		//缩回实时检测	
		IF (enablecloseAprSw AND NOT closeAprSw) AND closeRelay  THEN
			errorStep:=2;
		END_IF
		IF PVType=PVType_Other THEN
			;// 其他PV类型的关注点
		END_IF
	END_IF
END_IF
END_ACTION

ACTION VersionLog:
(*
版本: V1.0.0.0
说明:
	1. 首个版本
	2. 含普通PV类型的控制
	3. 可配置是否有到位信号, 以及到位稳定时间
(--------------------------------------------------)
新版本: V1.0.1.0
更新时间: 2019/11/20 19:00
更新说明:
	1. 优化编写方式
	2. 修改错误编码起始位，现改为从1开始
(--------------------------------------------------)
新版本: V1.0.1.1
更新时间: 2020/03/23 23:00
更新说明:
	1. 优化报错方式
	2. 增加打开、关闭、复位和停止触发函数
(--------------------------------------------------)
新版本: V1.0.1.2
更新时间: 2020/04/22 09:50
更新说明:
	1. 增加中文报警输出
(--------------------------------------------------)
新版本: V1.0.1.3
更新时间: 2020/09/16
更新说明:
	1. 开放错误ID、错误文本信息获取接口
(--------------------------------------------------)
新版本: V1.0.1.4
更新时间: 2020/10/06
更新说明:
	1. 移除控制模式变量，增加HMI启用条件
	2. 增加外部获取打开关闭完成信号接口函数
(--------------------------------------------------)
新版本: V1.0.1.5
更新时间: 2020/10/14
更新说明:
	1. 优化代码
(--------------------------------------------------)
*)
END_ACTION

END_FUNCTION_BLOCK

// ---- POUs/Communication/PLC_PDV.TcPOU
PROGRAM PLC_PDV
VAR_INPUT
	nSocketType:UINT:=0;// socket 类型; 0 表示 server; 1 表示 client;
	sTerminalName:STRING;// 通讯对方名称 自定义
	sHost:STRING(20):='127.0.0.1';// 通讯IP地址; server时表示本地host; client时表示远程host
	nPort:UDINT:=8900;// 通讯端口号;
	bEnable:BOOL:=TRUE;// 通讯启用\禁用连接
	sSendSuffix:STRING:='';//此处可统一添加发送后缀字符 $R$N
	nQueueInterval:UDINT:=50;// 发送队列时间间隔 单位ms
	logHandleArray:ARRAY [1..5] OF POINTER TO printLogModule_EX;// log 操作 handle 数组
	logHandleArrayLength:UINT:=0;// log 操作 handle 数组长度, 不超过5
	readStateFlag:BOOL;
	readPressureFlag:BOOL;
	readPostitionFlag:BOOL;
	readSetVal:BOOL;
	pvCloseCommunication		:BOOL;// PVClose
	pvOpenCommunication			:BOOL;// PVOpen
	pvPosOrPreCommunication		:BOOL;// PV Pos:=false;Pressure:True;
	pvReadPos:INT;// 位置
	pvReadPre:INT;// 压力
END_VAR
VAR_OUTPUT
	bSendCondition	:BOOL;//可发送条件
	bSocketConnected:BOOL;//连接状态
END_VAR
VAR CONSTANT
	cNumBegin		:DINT:=1;
	cNumEnd			:DINT:=100;
END_VAR
VAR
	sendDataArray	:ARRAY [cNumBegin..cNumEnd] OF STRING(255);
	length			:DINT:=0;
	endPoint		:DINT:=cNumBegin;
	popupSendData	:STRING(255);
	//popup
	popupStep		:UINT:=0;
	popupTON1		:TON;
	popupTON2		:TON;
	iPopup			:DINT:=0;
	_PopupLength	:DINT:=0;
END_VAR
VAR
	tcpipClient					:tcpipClientModule_EX;
	tcpipServer					:tcpipServerModule_EX;////定义服务器对象
	
	tcpipSendDataBuff_Server	:STRING(255);//发送数据 Buff server
	tcpipSendDataBuff_Client	:STRING(255);//发送数据 Buff client
	
	tcpipSendDataClear			:STRING(255);//发送数据 清空
	tcpipSendData				:STRING(255);//发送数据
	
	tcpipRecDataBuff_Server		:STRING(255);//已接收数据 Buff server
	tcpipRecDataBuff_Client		:STRING(255);//已接收数据 Buff client
	
	tcpipRecDataClear			:STRING(255);//已接收数据 清空
	tcpipRecData				:STRING(255);//已接收数据
	
	tcpConnectR_Trig			:R_Trig;//初始连接上升沿
	tcpConnectF_Trig			:F_Trig;//初始连接下降沿
	registerStep				:UDINT;//ALC注册控制步
	registerTON					:TON;//ALC注册延时
	
	logHandleArray_index		:UINT:=1;
END_VAR
VAR
	bTrig_Start:BOOL;
	rTrig_Start:R_TRIG;
	tTrig_Start:TON;
	
	bTrig_Stop:BOOL;
	rTrig_Stop:R_TRIG;
	tTrig_Stop:TON;
	
	bTrig_Reset:BOOL;
	rTrig_Reset:R_TRIG;
	tTrig_Reset:TON;
	
	
	bTrig_Init:BOOL;
	rTrig_Init:R_TRIG;
	
	bTrig_All_Home:BOOL;
	rTrig_All_Home:R_TRIG;
	
	bTrig_Z_Safe:BOOL;
	rTrig_Z_Safe:R_TRIG;
	
	bTrig_P_Pos_:BOOL;
	rTrig_P_Pos_:R_TRIG;
	nTrig_P_Pos_TrayNum:UINT:=1;
	nTrig_P_Pos_RowNum:UINT:=1;
	
	bTrig_Move_P_:BOOL;
	rTrig_Move_P_:R_TRIG;
	nTrig_Move_P_TrayNum:UINT:=1;
	nTrig_Move_P_RowNum:UINT:=1;
	nTrig_Move_P_PosNum:UINT:=1;
	findposstart	:INT;
	findposend		:INT;
	find_pos		:INT;
	recStrTemp		:STRING(255);
END_VAR


CASE nSocketType OF
0://TCPIP server
	tcpipServer(
		sSrvNetId:= , 
		sLocalHost:=sHost , 
		nLocalPort:=nPort , 
		bStartConnect:=bEnable , 
		tcpipSDataLen:=TO_UDINT(LEN(tcpipSendDataBuff_Server)) , 
		tcpipSData:=ADR(tcpipSendDataBuff_Server) , 
		bSend:= , 
		tcpipRecDataLen:=SIZEOF(tcpipRecDataBuff_Server) , 
		tcpipRecData:=ADR(tcpipRecDataBuff_Server) , 
		bAccepted=> , 
		bSendBusy=> , 
		bRecData=> );
	bSendCondition:=tcpipServer.bAccepted AND NOT tcpipServer.bSendBusy;
	//TCPIP连接
	bSocketConnected:=tcpipServer.bAccepted;
	IF NOT tcpipServer.bAccepted THEN
		length:=0;
		endPoint:=cNumBegin;
	END_IF
	tcpConnectR_Trig(CLK:=tcpipServer.bAccepted);
	tcpConnectF_Trig(CLK:=tcpipServer.bAccepted);

1://TCPIP client
	tcpipClient(
		sSrvNetId:= , 
		sRemoteHost:=sHost , 
		nRemotePort:=nPort , 
		bStartConnect:=bEnable , 
		tcpipSDataLen:=TO_UDINT(LEN(tcpipSendDataBuff_Client)) , 
		tcpipSData:=ADR(tcpipSendDataBuff_Client) , 
		bSend:= , 
		tcpipRecDataLen:=SIZEOF(tcpipRecDataBuff_Client) , 
		tcpipRecData:=ADR(tcpipRecDataBuff_Client) , 
		bConnected=> , 
		bSendBusy=> , 
		bRecData=> );
	bSendCondition:=tcpipClient.bConnected AND NOT tcpipClient.bSendBusy;
	//TCPIP连接
	bSocketConnected:=tcpipClient.bConnected;
	IF NOT tcpipClient.bConnected THEN
		length:=0;
		endPoint:=cNumBegin;
	END_IF
	tcpConnectR_Trig(CLK:=tcpipClient.bConnected);
	tcpConnectF_Trig(CLK:=tcpipClient.bConnected);
END_CASE

IF tcpConnectR_Trig.Q THEN
	FOR logHandleArray_index:=1 TO logHandleArrayLength DO
		logHandleArray[logHandleArray_index]^.append(CONCAT(sTerminalName, ' has been connected'));
	END_FOR
	registerStep:=10;
END_IF
IF tcpConnectF_Trig.Q THEN
	FOR logHandleArray_index:=1 TO logHandleArrayLength DO
		logHandleArray[logHandleArray_index]^.append(CONCAT(sTerminalName, ' has been disconnected'));
	END_FOR
	registerStep:=0;
END_IF
//数据接收处理
CASE nSocketType OF
0://TCPIP server
	IF tcpipServer.bRecData THEN
		tcpipRecData:=tcpipRecDataBuff_Server;//buff转存
		tcpipRecDataBuff_Server:=tcpipRecDataClear;//转存之后清空buff
		dataProcessing();
	END_IF
1://TCPIP client
	IF tcpipClient.bRecData THEN
		tcpipRecData:=tcpipRecDataBuff_Client;//buff转存
		tcpipRecDataBuff_Client:=tcpipRecDataClear;//转存之后清空buff
		dataProcessing();
	END_IF
END_CASE


popup();

CASE registerStep OF
0:
	//Ready
END_CASE

METHOD appendSend : BOOL
VAR_INPUT
	str			:STRING(255);
END_VAR
VAR
	suffix					:STRING;
	strTemp_appendSend		:STRING(255);
END_VAR

IF endPoint>(cNumEnd-1) THEN
	RETURN;
END_IF
suffix:=sSendSuffix;//此处可统一添加发送后缀字符 $R$N

strTemp_appendSend:=CONCAT(str,suffix);
sendDataArray[endPoint]:=strTemp_appendSend;

endPoint:=endPoint+1;
length:=endPoint-cNumBegin;
END_METHOD

METHOD dataProcessing : BOOL
VAR_INPUT
END_VAR
VAR
END_VAR
FOR logHandleArray_index:=1 TO logHandleArrayLength DO
	CASE nSocketType OF
	0://TCPIP server
	//	logHandleArray[logHandleArray_index]^.append(CONCAT(CONCAT(CONCAT('Recevie From ', sTerminalName), ' -- '),tcpipRecData));
	1://TCPIP client
	//	logHandleArray[logHandleArray_index]^.append(CONCAT(CONCAT(CONCAT('Recevie From ', sTerminalName), ' -- '),tcpipRecData));
	END_CASE
END_FOR
findposend:=0;
find_pos:=0;
IF MID(tcpipRecData,4,1)='i:30' THEN
	readStateFlag:=TRUE;
	CASE STRING_TO_INT(MID(tcpipRecData,1,6)) OF // 2:Pos 3:Close 4:Open 5:Pressur 6:Hold 7:Learn 8:interlock Open 9:interLock Closed
		2:
			pvPosOrPreCommunication:=FALSE;
			pvCloseCommunication:=FALSE;
			pvOpenCommunication:=FALSE;
		3:
			pvPosOrPreCommunication:=FALSE;
			pvCloseCommunication:=TRUE;
			pvOpenCommunication:=FALSE;
		4:
			pvPosOrPreCommunication:=FALSE;
			pvCloseCommunication:=FALSE;
			pvOpenCommunication:=TRUE;
		5:
			pvPosOrPreCommunication:=TRUE;
			pvCloseCommunication:=FALSE;
			pvOpenCommunication:=FALSE;
		ELSE
			pvPosOrPreCommunication:=FALSE;
			pvCloseCommunication:=FALSE;
			pvOpenCommunication:=FALSE;
	END_CASE
END_IF
IF MID(tcpipRecData,2,1)='A:' THEN
	readPostitionFlag:=TRUE;
	pvReadPos:=STRING_TO_INT(MID(tcpipRecData,6,3));
END_IF
IF MID(tcpipRecData,2,1)='P:' THEN
	readPressureFlag:=TRUE;
	pvReadPre:=STRING_TO_INT(MID(tcpipRecData,8,3));
	IF pvReadPre<0 THEN
		pvReadPre:=0;
	END_IF
END_IF
END_METHOD

METHOD PRIVATE popup : BOOL
VAR_INPUT
END_VAR
CASE popupStep OF
0:
	IF length>0 AND bSendCondition THEN
		_PopupLength:=length;
		popupSendData:=sendDataArray[cNumBegin];
		FOR iPopup:=cNumBegin TO (_PopupLength-1) DO
			sendDataArray[iPopup]:=sendDataArray[iPopup+1];
		END_FOR
		endPoint:=endPoint-1;
		length:=endPoint-cNumBegin;
		sendData(popupSendData);//此处是调用信息发送
		popupStep:=10;
	END_IF
10:
	popupTON2(IN:=NOT popupTON2.Q, PT:=T#2S);
	IF NOT bSendCondition OR popupTON2.Q THEN
		popupTON2(IN:=FALSE);
		popupStep:=11;
	END_IF
11:
	IF bSendCondition THEN
		popupStep:=12;
	END_IF
	popupTON1(IN:=FALSE);
12:
	//popupTON1(IN:=NOT popupTON1.Q,PT:=T#10MS);
	popupTON1(IN:=NOT popupTON1.Q,PT:=TO_TIME(nQueueInterval));
	IF popupTON1.Q THEN
		popupStep:=0;
	END_IF
END_CASE
END_METHOD

METHOD ReadPosition : BOOL
VAR_INPUT
END_VAR
VAR
END_VAR
appendSend('A:$N');
END_METHOD

METHOD ReadPressure : BOOL
VAR_INPUT
END_VAR
VAR
END_VAR
appendSend('P:$N');
END_METHOD

METHOD ReadSetVal : BOOL
VAR_INPUT
END_VAR
VAR
END_VAR
appendSend('i:38$N');
END_METHOD

METHOD ReadState : BOOL
VAR_INPUT
END_VAR
VAR
END_VAR
appendSend('i:30$N');
END_METHOD

METHOD PRIVATE sendData : BOOL
VAR_INPUT
	dataStruct	:STRING(255);
END_VAR
IF bSendCondition AND bEnable THEN
	tcpipSendData:=dataStruct;
	
	CASE nSocketType OF
	0://TCPIP server
		tcpipSendDataBuff_Server:=tcpipSendData;
		tcpipSendData:=tcpipSendDataClear;	
		tcpipServer.bSend:=TRUE;
	1://TCPIP client
		tcpipSendDataBuff_Client:=tcpipSendData;
		tcpipSendData:=tcpipSendDataClear;	
		tcpipClient.bSend:=TRUE;
	END_CASE
	
	FOR logHandleArray_index:=1 TO logHandleArrayLength DO
		CASE nSocketType OF
		0://TCPIP server
			//logHandleArray[logHandleArray_index]^.append(CONCAT(CONCAT(CONCAT('Send To ', sTerminalName), ' -- '),tcpipSendDataBuff_Server));
		1://TCPIP client
			//logHandleArray[logHandleArray_index]^.append(CONCAT(CONCAT(CONCAT('Send To ', sTerminalName), ' -- '),tcpipSendDataBuff_Client));
		END_CASE
	END_FOR
END_IF
END_METHOD

METHOD WriteAccessMode : BOOL
VAR_INPUT
	mode:INT;// 0:Local  1:Remote  2:锁定远程操作，无法通过服务端口更改为本地
END_VAR
CASE mode OF
	0:
		appendSend('c:0100$N');
	1:
		appendSend('c:0101$N');
	2:
		appendSend('c:0102$N');
	ELSE
		appendSend('c:0102$N');
END_CASE
END_METHOD

METHOD WriteCloseValve : BOOL
VAR_INPUT

END_VAR
VAR

END_VAR

appendSend('C:$N');
END_METHOD

METHOD WriteHold : BOOL
VAR_INPUT
END_VAR
appendSend('O:$N');
END_METHOD

METHOD WriteLearn : BOOL
VAR_INPUT
	positon:REAL;
	point:INT;
END_VAR
VAR
	intTemp:DINT;
	intTemp1:DINT;
	intTemp2:DINT;
	intTemp3:DINT;
	intTemp4:DINT;
	intTemp5:DINT;
	intTemp6:DINT;
	intTemp7:DINT;
	intTemp8:DINT;
	str:STRING;
END_VAR
str:='L:';
intTemp:=LREAL_TO_DINT(positon*EXPT(10,point));
intTemp8:=LREAL_TO_INT(FLOOR(intTemp/10000000));
str:=CONCAT(str,DINT_TO_STRING(intTemp8));
intTemp7:=LREAL_TO_INT(FLOOR(intTemp/1000000 MOD 10));
str:=CONCAT(str,DINT_TO_STRING(intTemp7));
intTemp6:=LREAL_TO_INT(FLOOR(intTemp/100000 MOD 10));
str:=CONCAT(str,DINT_TO_STRING(intTemp6));
intTemp5:=LREAL_TO_INT(FLOOR(intTemp/10000 MOD 10));
str:=CONCAT(str,DINT_TO_STRING(intTemp5));
intTemp4:=LREAL_TO_INT(FLOOR(intTemp/1000 MOD 10));
str:=CONCAT(str,DINT_TO_STRING(intTemp4));
intTemp3:=LREAL_TO_INT(FLOOR(intTemp/100 MOD 10));
str:=CONCAT(str,DINT_TO_STRING(intTemp3));
intTemp2:=LREAL_TO_INT(FLOOR(intTemp/10 MOD 10));
str:=CONCAT(str,DINT_TO_STRING(intTemp2));
intTemp1:=LREAL_TO_INT(FLOOR(intTemp MOD 10));
str:=CONCAT(str,DINT_TO_STRING(intTemp1));
str:=CONCAT(str,'$N');
appendSend(str);
END_METHOD

METHOD WriteOpenValve : BOOL
VAR_INPUT
END_VAR
appendSend('O:$N');
END_METHOD

METHOD WritePositionControl : BOOL
VAR_INPUT
	pressure:REAL;
	point:INT;
END_VAR
VAR
	intTemp:DINT;
	intTemp1:DINT;
	intTemp2:DINT;
	intTemp3:DINT;
	intTemp4:DINT;
	intTemp5:DINT;
	intTemp6:DINT;
	str:STRING;
END_VAR
str:='R:';
intTemp:=LREAL_TO_DINT(pressure*EXPT(10,point));
intTemp6:=LREAL_TO_INT(FLOOR(intTemp/100000 MOD 10));
str:=CONCAT(str,DINT_TO_STRING(intTemp6));
intTemp5:=LREAL_TO_INT(FLOOR(intTemp/10000 MOD 10));
str:=CONCAT(str,DINT_TO_STRING(intTemp5));
intTemp4:=LREAL_TO_INT(FLOOR(intTemp/1000 MOD 10));
str:=CONCAT(str,DINT_TO_STRING(intTemp4));
intTemp3:=LREAL_TO_INT(FLOOR(intTemp/100 MOD 10));
str:=CONCAT(str,DINT_TO_STRING(intTemp3));
intTemp2:=LREAL_TO_INT(FLOOR(intTemp/10 MOD 10));
str:=CONCAT(str,DINT_TO_STRING(intTemp2));
intTemp1:=LREAL_TO_INT(FLOOR(intTemp MOD 10));
str:=CONCAT(str,DINT_TO_STRING(intTemp1));
str:=CONCAT(str,'$N');
appendSend(str);
END_METHOD

METHOD WritePressureAlignment : BOOL
VAR_INPUT
	pressure:REAL;
	point:INT;
END_VAR
VAR
	intTemp:DINT;
	intTemp1:DINT;
	intTemp2:DINT;
	intTemp3:DINT;
	intTemp4:DINT;
	intTemp5:DINT;
	intTemp6:DINT;
	intTemp7:DINT;
	intTemp8:DINT;
	str:STRING;
END_VAR
str:='c:6002';
intTemp:=LREAL_TO_DINT(pressure*EXPT(10,point));
intTemp8:=LREAL_TO_INT(FLOOR(intTemp/10000000));
str:=CONCAT(str,DINT_TO_STRING(intTemp8));
intTemp7:=LREAL_TO_INT(FLOOR(intTemp/1000000 MOD 10));
str:=CONCAT(str,DINT_TO_STRING(intTemp7));
intTemp6:=LREAL_TO_INT(FLOOR(intTemp/100000 MOD 10));
str:=CONCAT(str,DINT_TO_STRING(intTemp6));
intTemp5:=LREAL_TO_INT(FLOOR(intTemp/10000 MOD 10));
str:=CONCAT(str,DINT_TO_STRING(intTemp5));
intTemp4:=LREAL_TO_INT(FLOOR(intTemp/1000 MOD 10));
str:=CONCAT(str,DINT_TO_STRING(intTemp4));
intTemp3:=LREAL_TO_INT(FLOOR(intTemp/100 MOD 10));
str:=CONCAT(str,DINT_TO_STRING(intTemp3));
intTemp2:=LREAL_TO_INT(FLOOR(intTemp/10 MOD 10));
str:=CONCAT(str,DINT_TO_STRING(intTemp2));
intTemp1:=LREAL_TO_INT(FLOOR(intTemp MOD 10));
str:=CONCAT(str,DINT_TO_STRING(intTemp1));
str:=CONCAT(str,'$N');
appendSend(str);
END_METHOD

METHOD WritePressureControl : BOOL
VAR_INPUT
	pressure:REAL;
	point:INT;
END_VAR
VAR
	intTemp:DINT;
	intTemp1:DINT;
	intTemp2:DINT;
	intTemp3:DINT;
	intTemp4:DINT;
	intTemp5:DINT;
	intTemp6:DINT;
	intTemp7:DINT;
	intTemp8:DINT;
	str:STRING;
END_VAR
str:='S:';
intTemp:=LREAL_TO_DINT(pressure*EXPT(10,point));
intTemp8:=LREAL_TO_INT(FLOOR(intTemp/10000000));
str:=CONCAT(str,DINT_TO_STRING(intTemp8));
intTemp7:=LREAL_TO_INT(FLOOR(intTemp/1000000 MOD 10));
str:=CONCAT(str,DINT_TO_STRING(intTemp7));
intTemp6:=LREAL_TO_INT(FLOOR(intTemp/100000 MOD 10));
str:=CONCAT(str,DINT_TO_STRING(intTemp6));
intTemp5:=LREAL_TO_INT(FLOOR(intTemp/10000 MOD 10));
str:=CONCAT(str,DINT_TO_STRING(intTemp5));
intTemp4:=LREAL_TO_INT(FLOOR(intTemp/1000 MOD 10));
str:=CONCAT(str,DINT_TO_STRING(intTemp4));
intTemp3:=LREAL_TO_INT(FLOOR(intTemp/100 MOD 10));
str:=CONCAT(str,DINT_TO_STRING(intTemp3));
intTemp2:=LREAL_TO_INT(FLOOR(intTemp/10 MOD 10));
str:=CONCAT(str,DINT_TO_STRING(intTemp2));
intTemp1:=LREAL_TO_INT(FLOOR(intTemp MOD 10));
str:=CONCAT(str,DINT_TO_STRING(intTemp1));
str:=CONCAT(str,'$N');
appendSend(str);
END_METHOD

METHOD WriteZero : BOOL
VAR_INPUT
		

END_VAR
appendSend('Z:$N');
END_METHOD

END_PROGRAM

// ---- POUs/BaseModule/TcpIpModule_EX/serverModule_EX/tcpipServerModule_EX.TcPOU
//可实现TCPIP Server 数据的收发
FUNCTION_BLOCK tcpipServerModule_EX
VAR_INPUT
	sSrvNetId			:T_AmsNetId:='';
	sLocalHost			:STRING(20):='';//服务器的IP地址
	nLocalPort			:UDINT:=5000;//服务器的端口号
	bStartConnect		:BOOL:=TRUE;//可实现外部控制服务器的重新连接
//Send
	tcpipSDataLen		:UDINT;//待发送数据长度--外部传递进来
	tcpipSData			:POINTER TO BYTE;//待发送数据源----外部以指针的形式传递进来
	bSend				:BOOL:=FALSE;//数据发送触发信号
//Receive
	tcpipRecDataLen		:UDINT;//已接收数据长度--外部传递进来
	tcpipRecData		:POINTER TO BYTE;//已接收数据源--外部以指针的形式传递进来(ADR函数)
END_VAR

VAR_OUTPUT
//Connect
	bAccepted			:BOOL:=FALSE;//表示客户端连接状态
//Send
	bSendBusy			:BOOL:=FALSE;//数据发送中
//Receive
	bRecData			:BOOL:=FALSE;//数据接收有效信号,上升沿有效
END_VAR

VAR
//Listen
	createStep			:UINT:=0;
	socketListenFB		:FB_SocketListen;(*TCP/IP Sever建立Listen功能块*)
	hListener			:T_HSOCKET;(*TCP/IP的监听句柄*)
	createDelayTime		:TIME:=T#500MS;
	createDelayTon		:TON;
	createCheckTime		:TIME:=T#1000MS;
	createCheckTon		:TON;
//Accept
	socketAcceptFB		:FB_SocketAccept;	(*TCP/IP Accept功能块*)
	hSocket				:T_HSOCKET;(*TCP/IP的句柄*)
//Send
	socketSendFB		:FB_SocketSend;	(*TCP/IP的Send功能块*)
	sendDataTempLen		:UDINT;//待发送数据缓存 长度
	sendDataTemp		:POINTER TO BYTE;//待发送数据缓存
	sendStep			:UINT:=0;
//Receive
	recStep				:UINT:=0;
	socketReceiveFB		:FB_SocketReceive;(*TCP/IP的Receive功能块*)
	recDelayTime		:TIME:=T#1S;
	recDelayTon			:TON;
//Close
	socketCloseFB		:FB_SocketClose;(*TCP/IP的Close连接的功能块*)	
END_VAR

create();
receive();
send();
socketCloseFB(
	sSrvNetId:=sSrvNetId,
	hSocket:=,
	bExecute:=FALSE);

METHOD ascii2String : STRING(g_nMaxByte_Server)
VAR_INPUT
	byteArr:ARRAY [1..g_nMaxByte_Server] OF BYTE;
END_VAR
VAR
	i:UINT;
	strTemp:STRING(g_nMaxByte_Server);
END_VAR
FOR i:=1 TO g_nMaxByte_Server DO
	strTemp:=concat(strTemp,F_ToCHR(c:=byteArr[i]));
END_FOR
ascii2string:=strTemp;
END_METHOD

METHOD PRIVATE close : BOOL
VAR_INPUT
END_VAR
//关闭hSocket这个端口的连接
socketCloseFB(
	sSrvNetId:=sSrvNetId,
	hSocket:=hSocket, 
	bExecute:=TRUE, 			//TCP/IP端口关闭的执行位
	tTimeout:=T#1S,
	bBusy=>,
	bError=>,
	nErrId=>);
socketCloseFB(
	sSrvNetId:=sSrvNetId,
	hSocket:=,
	bExecute:=FALSE);
hSocket.handle:=0;
bAccepted:=FALSE;
END_METHOD

METHOD PRIVATE closeListen : BOOL
VAR_INPUT
END_VAR
//关闭 监听 hListener 这个端口
socketCloseFB(
	sSrvNetId:=sSrvNetId,
	hSocket:=hListener, 
	bExecute:=TRUE, 			//TCP/IP端口关闭的执行位
	tTimeout:=,
	bBusy=>,
	bError=>,
	nErrId=>);
socketCloseFB(
	sSrvNetId:=sSrvNetId,
	hSocket:=,
	bExecute:=FALSE);
END_METHOD

METHOD PRIVATE create : BOOL
VAR_INPUT
END_VAR

VAR
END_VAR

CASE createStep OF
0:
	IF socketListenFB.bExecute OR bAccepted THEN
		RETURN;
	END_IF
	socketListenFB(
	   sSrvNetId:=sSrvNetId,
	   sLocalHost:=sLocalHost,
	   nLocalPort:=nLocalPort,
	   bExecute:=FALSE);
	socketCloseFB(
		sSrvNetId:=sSrvNetId,
		hSocket:=hListener, 
		bExecute:=TRUE, 			//TCP/IP端口关闭的执行位
		tTimeout:=T#1S,
		bBusy=>,
		bError=>,
		nErrId=>);
	createStep:=createStep+1;
1:
	createStep:=createStep+1;
2:
	createStep:=createStep+1;
3:
	socketListenFB(
		sSrvNetId:=sSrvNetId,
		sLocalHost:=sLocalHost,
		nLocalPort:=nLocalPort,
		bExecute:=TRUE,
		tTimeout:=T#1S,
		bBusy=>,
		bError=>,
		nErrId=>,
		hListener=>hListener);
	IF NOT socketListenFB.bBusy THEN
		IF socketListenFB.bError (*AND socketListenFB.nErrId<>32771*)THEN
			createStep:=createStep+1;
		ELSE
			//Listen
			createStep:=50;
			socketAcceptFB(
				sSrvNetId:=sSrvNetId,
				hListener:=hListener,		//TCP/IP的监听句柄
				bExecute:=FALSE);	
		END_IF
	END_IF
	createDelayTon(IN:=FALSE);

4://delay
	createDelayTon(IN:=NOT createDelayTon.Q ,PT:=createDelayTime);
	IF createDelayTon.Q THEN
		createDelayTon(IN:=FALSE);
		createStep:=createStep+1;
		socketListenFB(
			sSrvNetId:=sSrvNetId,
			sLocalHost:=sLocalHost,
			nLocalPort:=nLocalPort,
			bExecute:=FALSE);
	END_IF
5:
	createStep:=0;
	close();
	
50:	
	createStep:=51;
	close();
51:
	socketAcceptFB(
		sSrvNetId:=sSrvNetId, 
		hListener:=hListener,//TCP/IP的监听句柄
		bExecute:=TRUE,//TCP/IP接受连接请求的执行位
		tTimeout:=T#1S, 
		bAccepted=>bAccepted,
		bBusy=> , 
		bError=> , 
		nErrId=> , 
		hSocket=>hSocket );//获取的TCP/IP句柄 AND socketAcceptFB.bBusy
	IF (bAccepted AND hSocket.handle<>0) (*OR NOT bStartConnect*) THEN
		socketListenFB(
			sSrvNetId:=sSrvNetId,
			sLocalHost:=sLocalHost,
			nLocalPort:=nLocalPort,
			bExecute:=FALSE);
		createStep:=100;
	END_IF
	IF NOT bStartConnect THEN
		close();
		createStep:=100;
	END_IF
	socketAcceptFB(
		sSrvNetId:=sSrvNetId,
		hListener:=hListener,
		bExecute:=FALSE);
	createCheckTon(IN:=FALSE);

100:
	createCheckTon(IN:=NOT bAccepted OR NOT bStartConnect, PT:=createCheckTime);
	IF createCheckTon.Q THEN
		createStep:=50;
		createCheckTon(IN:=FALSE);
	END_IF
END_CASE
END_METHOD

METHOD PRIVATE receive : BOOL
VAR_INPUT
END_VAR
VAR
	recDataClear		:POINTER TO BYTE;//已接收数据源--外部以指针的形式传递进来(ADR函数)
END_VAR

CASE recStep OF
0:
	IF hSocket.handle>0 AND bAccepted THEN
		recStep:=10;
	END_IF

10:
	bRecData:=FALSE;
	socketReceiveFB(
			sSrvNetId:=sSrvNetId,
			hSocket:=hSocket,
			cbLen:= tcpipRecDataLen,
			pDest:= tcpipRecData,
			bExecute:= TRUE,
			tTimeout:=T#1S,
			bBusy=>,
			bError=>,
			nErrId=>,
			nRecBytes=>);
	
	IF (NOT socketReceiveFB.bBusy) THEN
		recStep:=20;
	END_IF
20:
	socketReceiveFB(sSrvNetId:=sSrvNetId,hSocket:=hSocket,bExecute :=FALSE);
	IF (NOT socketReceiveFB.bBusy) THEN
		IF (socketReceiveFB.bError) THEN
			close();//关闭socket
			recStep:=110;
		ELSE
			IF socketReceiveFB.nRecBytes>0 THEN
				tcpipRecData:=recDataClear;//清空缓存数据
				bRecData:=TRUE;
			END_IF
			recStep:=10;//继续接收通道数据
		END_IF
	END_IF

110:
	recDelayTon(IN:=NOT recDelayTon.Q ,PT:=recDelayTime);
	IF recDelayTon.Q THEN
		recDelayTon(IN:=FALSE);
		recStep:=recStep+10;
	END_IF
120:
	recStep:=0;	
END_CASE
END_METHOD

METHOD PRIVATE send : BOOL
VAR_INPUT
END_VAR

VAR
END_VAR

CASE sendStep OF
0:
	IF bAccepted THEN
		bSendBusy:=FALSE;
		socketSendFB(hSocket:=hSocket,bExecute :=FALSE);
		IF bSend THEN
			sendStep:=10;
			sendDataTempLen:=tcpipSDataLen;
			sendDataTemp:=tcpipSData;
			bSendBusy:=TRUE;
			bSend:=FALSE;
		END_IF
	END_IF
10:
	socketSendFB(
			sSrvNetId:=sSrvNetId, 
			hSocket:=hSocket , 
			cbLen:= sendDataTempLen,
			pSrc:= sendDataTemp, 
			bExecute:= TRUE,
			tTimeout:= T#1S, 
			bBusy=> , 
			bError=> , 
			nErrId=> );
	
	IF NOT socketSendFB.bBusy THEN
		sendStep:=sendStep+10;
	END_IF
20:
	sendStep:=sendStep+10;
30:
	bSendBusy:=FALSE;
	bSend:=FALSE;
	sendStep:=0;
END_CASE
END_METHOD

METHOD string2ASCII : ARRAY [1..g_nMaxByte_Server] OF BYTE
VAR_INPUT
	str:STRING(g_nMaxByte_Server);
END_VAR
VAR
	i:DINT;
	byteTemp:ARRAY [1..g_nMaxByte_Server] OF BYTE;
	strB:STRING(1);
	strTemp:STRING(g_nMaxByte_Server);
END_VAR

strTemp:=str;
FOR i:=1 TO g_nMaxByte_Server DO
	strB:=LEFT(strTemp,1);
	strTemp:=DELETE(strTemp,1,1);
	byteTemp[i]:=F_ToASC(str:=strB);
END_FOR
string2ASCII:=byteTemp;
END_METHOD

ACTION VersionLog:
(*
版本: V1.0.0.0
说明:
	1. 首个版本
(**************************************************)
版本: V1.0.0.1
说明:
	1. 更新close函数，关闭连接后清零连接句柄
(**************************************************)
版本: V1.0.0.2
说明:
	1. 更新cread函数，处理无法接受新连接的bug
(**************************************************)
*)
END_ACTION

END_FUNCTION_BLOCK

// ---- POUs/BaseModule/ActionModule/RFModule/RFModule.TcPOU
(*
--报错编号0: 无报错
--报错编号1: openend Error
--报错编号2: close Error
*)
FUNCTION_BLOCK RFModule
VAR_IN_OUT
	WarmHMI					:WARMStruct;
	NoteHMI					:NoteStruct;
	operatorLog				:printLogModule_EX;
END_VAR
VAR_INPUT
	HMIItf						:RFHMIStruts;// 每个RF对象都关联了一个HMI
	RFTYPE						:RFType:=RFType_Default;// 设置RF的类型
	real_TimeMonitor			:BOOL:=TRUE;//实时状态检测
	co_control					:BOOL;// 共同计时
	open						:BOOL:=FALSE;//启动触发信号
	openCondition				:BOOL:=TRUE;//启动条件
	close						:BOOL:=FALSE;//停止触发信号
	closeCondition				:BOOL:=TRUE;//停止条件
	reset						:BOOL:=FALSE;//复位信号
	readCondition				:BOOL:=TRUE;//读取条件
	stop						:BOOL:=FALSE;//停止信号
	power						:BOOL:=TRUE;// RF动作后是否关闭继电器得电状态, TRUE--保持得电,FALSE--断开得电
	enable						:BOOL:=TRUE;// RF禁用条件
	//ctrlMode					:ControlMode:=ControlMode.eManualCtrMode;//eManualCtrMode or eAutoCtrMode
	hmiEN						:BOOL:=TRUE;//HMI 启用条件
	serialExcute				:BOOL;// RS485、232开始一次参数读取
	
	errorDelayTime				:TIME:=T#100S;//分子泵感应器感应超时
	
	ACCMaxtime					:TIME:=T#20S;// RF加速最大时间 启动过程
	DCCMaxtime					:TIME:=T#20S;// RF减速最大时间 停止过程
	
	doneDelayTimeShortopenend	:TIME:=T#100MS;//  RF启动感应到位延时_伸出
	doneDelayTimeShortcloseract	:TIME:=T#50MS;//  RF感应到位延时_收回
	doneDelayTimeLongopenend	:TIME:=T#500MS;//  RF感应到位延时_伸出
	doneDelayTimeLongcloseract	:TIME:=T#50MS;// RF感应到位延时_收回
	errorID						:UDINT:=0;// RF错误报警分配的起始ID
	nameTXT						:STRING(255):='';// RF名字
	
	AlmAprSw					:BOOL:=FALSE;// RF报警感应器信号,需要链接到实际的IO点
	ErrorAprSw					:BOOL:=FALSE;// RF报错感应器信号,需要链接到实际的IO点
	enableOpenAprSw				:BOOL:=TRUE;// 启用启动感应器,针对只有一个传感器的 RF
	enableCloseAprSw			:BOOL:=TRUE;// 启用停止感应器,针对只有一个传感器的 RF
	runTime						: LINT;// 运行时间
	mainPower					:BOOL;// RF主电源
	temperature					:REAL;// RF温度
	current						:REAL;// RF电流
	vol							:REAL;// RF电压
	serialSlaveID				:UINT;// RF ID
	serialError					:BOOL;// RF通讯错误
	setpower					:UDINT;// 设定功率	
	settime						:UDINT;// 设定时间
	noteWTXT_open				:WSTRING(255):="";// RF打开动作NoteTXT 中文
	noteWTXT_close				:WSTRING(255):="";// RF关闭动作NoteTXT 中文
	controlMode					:INT:=0;// 0 手动，1 Analog，2 RS232
	outputMode					:INT:=0;// 0 continuous，1 pulse
	outputState					:INT:=0;// 0 Stop,1 Start
	alarmState					:INT:=0;// 0 No Error,1 Error
	setpowerRead				:UDINT:=0;// 读取设置的功率值
	forwardpower				:UDINT;// 实际功率	
	reflectedpower				:UDINT;// 反馈功率
	maxpower					:UDINT;// 设置的最大功率值
END_VAR
VAR_OUTPUT
	note_open				:BOOL;// 开条件不满足提示
	note_close				:BOOL;// 关条件不满足提示
	openRelay				:BOOL:=FALSE;// RF启动执行继电器,需要链接到实际的IO点
	closeRelay				:BOOL:=FALSE;// RF停止执行继电器,需要链接到实际的IO点
	resetRelay				:BOOL:=FALSE;// RF复位执行继电器,需要链接到实际的IO点	
	rematime				:UDINT;// 剩余时间
	busy					:BOOL;// RFusy状态
	openbusy				:BOOL;// RF开动作Busy状态
	closebusy				:BOOL;// RF关动作Busy状态
	readbusy				:BOOL;// RF循环读取Busy状态
	done					:BOOL;// RF动作Done状态
	readdone					:BOOL;// RF动作Done状态
	opendone				:BOOL;// RF动作伸出完成
	closedone				:BOOL;// RF动作收回完成
	setpointdone			:BOOL;
	readerror			    :BOOL;// RF动作error状态
	error					:BOOL;// RF动作error状态
	errID					:UDINT;// RF动作errID
	errTXT					:STRING(255):='';// RF动作errTXT
	errWTXT					:WSTRING(255):="";// RF动作errTXT 中文
END_VAR
	
VAR	
	readAndWriteLock:BOOL;
	runTON					: TON;
	openErrorDelayTon		:Ton;
	openDoneDelayTon		:Ton;
	closeErrorDelayTon		:Ton;
	closeDoneDelayTon		:Ton;
	
	extendTrigRAlc			:R_Trig;//上升沿触发
	runTimeClearR			:R_Trig;//上升沿触发
	
	openendTrigRAlc			:R_Trig;//上升沿触发
	
	singleControltempR			:R_Trig;//上升沿触发
	singleControlR			:R_Trig;//上升沿触发
	singleControlF			:F_Trig;//上升沿触发
	
	openendTrigR1			:R_Trig;//上升沿触发
	openendTrigR1_Aiko		:R_Trig;//上升沿触发
	closeractTrigR1			:R_Trig;//上升沿触发
	resetTrigR1				:R_Trig;//上升沿触发
	stopTrigR1				:R_Trig;//上升沿触发
	powerTrigR1				:R_Trig;//上升沿触发
	
	openStep				:UINT:=0;
	closeStep				:UINT:=0;
	errorStep				:UINT:=0;
	readStep				:UINT:=0;
	
	resetRelayTON			:TON;
	resetRelayTONTime		:TIME:=T#2S;
	
	writeStep				:UINT:=0;
	writeMaxStep			:UINT:=0;
	
	notBusyMonitorDelayTon:TON;//动作不切换时，延迟检测
	notBusyMonitorDelayTime:TIME:=T#2S;//动作不切换延迟检测时间
	firstPower			    :BOOL:=TRUE;//首次上电标志位
	firstPowerTON			:TON;
	AccFTrig:F_TRIG;//检测加速信号下降延
	NormalRTrig:R_TRIG;//匀速上升沿
	DccFTrig:F_TRIG;// 检测减速信号下降延
	noteTON_P:tON;            // 操作提示标志位延时继电器
	noteTON_N:tON;            // 操作提示标志位延时继电器
	noteRTrig_P:R_TRIG;          // 操作提示
	noteRTrig_N:R_TRIG;          // 操作提示
	powerTon:TON;
	readTon1:TON;
	readTon2:TON;
	readTon3:TON;
	t1:TON;
	t2:TON;
	writeTON:TON;
	writeMaxTON:TON;
	readTON:TON;
	readErrorTimes:UINT:=0;
END_VAR

Init_ACT();
Error_ACT();
Open_ACT();
Close_ACT();
Reset_ACT();
Error_ACT();
Read_ACT();
WritePower_ACT();
WriteMaxPower_ACT();

(*
触发缩回动作，成功触发返回TRUE，触发失败返回FALSE
*)
METHOD Act_Close : BOOL
VAR_INPUT
END_VAR
IF enable AND closeCondition THEN// AND NOT busy
	Act_Close:=close:=TRUE;
ELSE
	Act_Close:=FALSE;
END_IF
END_METHOD

(*
触发伸出动作，成功触发返回TRUE，触发失败返回FALSE
*)
METHOD Act_Open : BOOL
VAR_INPUT
END_VAR
IF enable AND openCondition THEN// AND NOT busy
	Act_Open:=open:=TRUE;
ELSE
	Act_Open:=FALSE;
END_IF
END_METHOD

(*
触发复位报警动作，成功触发返回TRUE，触发失败返回FALSE
*)
METHOD Act_Reset : BOOL
VAR_INPUT
END_VAR
Act_Reset:=reset:=TRUE;
END_METHOD

(*
触发发送动作，成功触发返回TRUE，触发失败返回FALSE
*)
METHOD Act_SerialSend : BOOL
VAR_INPUT
END_VAR
IF TRUE THEN
	Act_SerialSend:=serialExcute:=TRUE;
ELSE
	Act_SerialSend:=FALSE;
END_IF
END_METHOD

METHOD Act_SetPoint : BOOL
VAR_INPUT
	setpoint:UDINT;
	_settime:UDINT;
	con_ctr:BOOL;
END_VAR
VAR_OUTPUT
	outTime:UDINT;
END_VAR
setpower:=HMIItf.setpower:=setpoint;
settime:=HMIItf.settime:=outTime:=_settime;
co_control:=con_ctr;
Act_Open();
END_METHOD

(*
触发停止输出动作，成功触发返回TRUE，触发失败返回FALSE
*)
METHOD Act_Stop : BOOL
VAR_INPUT
END_VAR
Act_Stop:=stop:=TRUE;
END_METHOD

(*
触发缩回动作，成功触发返回TRUE，触发失败返回FALSE
*)
METHOD Act_Write : BOOL
VAR_INPUT
END_VAR
IF writeStep<10 AND NOT readAndWriteLock THEN
	writeStep:=10;
	readAndWriteLock:=TRUE;
END_IF
END_METHOD

(*
触发缩回动作，成功触发返回TRUE，触发失败返回FALSE
*)
METHOD Act_Write_1 : BOOL
VAR_INPUT
END_VAR
IF writeStep<10 AND readAndWriteLock THEN
	writeStep:=10;
	readAndWriteLock:=TRUE;
END_IF
END_METHOD

ACTION Close_ACT:
//分子泵--close 触发
IF close AND NOT closeCondition THEN
	note_open:=FALSE;
	note_close:=TRUE;
	NoteHMI.showFlag:=TRUE;
	NoteHMI.showText:='';
	NoteHMI.showText:=CONCAT(NoteHMI.showText,nameTXT);
	NoteHMI.showText:=CONCAT(NoteHMI.showText,' Close Condition Not Satisfied!');
	operatorLog.append(CONCAT(nameTXT,' Close Not Done '));
END_IF
IF close AND enable AND closeCondition AND closeStep<20 THEN// AND NOT busy
	note_open:=FALSE;
	note_close:=FALSE;
	busy:=TRUE;
	writeStep:=0;
	writeMaxStep:=0;
	closebusy:=TRUE;
	openbusy:=FALSE;
	open:=FALSE;
	// searial_send(0)**************************************
	opendone:=FALSE;
	closedone:=FALSE;
	openStep:=0;
	closeStep:=10;
	readAndWriteLock:=TRUE;
	PLC_PowerRF.WriteStop();
	operatorLog.append(CONCAT(nameTXT,' Close Done '));
	//errorStep:=0;
END_IF
close:=FALSE;

CASE closeStep OF
0:
	//ready
	
10:
	IF readStep<10 AND writeStep<10 AND writeMaxStep<10 THEN
		closeErrorDelayTon(IN:=FALSE);
		closeDoneDelayTon(IN:=FALSE);
		closeRelay:=TRUE;
		PLC_PowerRF.WriteStop();
		openRelay:=FALSE;
		closeStep:=15;
		t2(IN:=FALSE);
	END_IF
15:
	t2(IN:=TRUE,PT:=T#0.2S);
	IF t2.Q THEN
		t2(IN:=FALSE);
		readAndWriteLock:=FALSE;
		PLC_PowerRF.WriteStop();
		closeStep:=20;
		busy:=FALSE;
	END_IF
20:// DCC与ACC一样，只不过ACC在Open逻辑；DCC 在Close逻辑里；  DCC=forwardpower<setpoint
	closeErrorDelayTon(IN:=(NOT (forwardpower=0 AND reflectedpower=0 AND rematime=0)),PT:=errorDelayTime);
	IF closeErrorDelayTon.Q THEN
		//done:=FALSE;
		opendone:=FALSE;
		closedone:=FALSE;
		errorStep:=2;
		closeStep:=40;
		RETURN;
	END_IF
	IF enablecloseAprSw THEN
		closeDoneDelayTon(IN:=(forwardpower=0 AND reflectedpower=0 AND rematime=0),PT:=doneDelayTimeShortcloseract);
	END_IF
	IF closeDoneDelayTon.Q THEN
		closeErrorDelayTon(IN:=FALSE);
		closeDoneDelayTon(IN:=FALSE);
		closeStep:=30;
	END_IF
30:
	busy:=FALSE;
	closebusy:=FALSE;
	openbusy:=FALSE;
	//done:=TRUE;
	opendone:=FALSE;
	closedone:=TRUE;
	errorStep:=0;
	closeStep:=0;
	readAndWriteLock:=FALSE;
	t2(IN:=FALSE);
40:
	busy:=FALSE;
	closebusy:=FALSE;
	openbusy:=FALSE;
	closeStep:=0;
	readAndWriteLock:=FALSE;
	t2(IN:=FALSE);
END_CASE
END_ACTION

ACTION Error_ACT:
CASE errorStep OF
	0:
		error:=FALSE;
		errID:=0;
		errTXT:='';
 (*
	1:
		error:=TRUE;
		errID:=errorID+errorStep;
		errTXT:=CONCAT(STR1:=nameTXT,STR2:=' Extend Error!');
		errWTXT:=WCONCAT(STR1:=TO_WSTRING(nameTXT),STR2:=" 伸出(打开)错误");
	2:
		error:=TRUE;
		errID:=errorID+errorStep;
		errTXT:=CONCAT(STR1:=nameTXT,STR2:=' Retract Error!');
		errWTXT:=WCONCAT(STR1:=TO_WSTRING(nameTXT),STR2:=" 缩回(关闭)错误");
		*)
	1..6:
		error:=TRUE;
		errID:=getErrID(errorStep);
		errTXT:=getErrTXT(errorStep);
		errWTXT:=getErrWTXT(errorStep);
END_CASE
END_ACTION

METHOD Get_Done_Close : BOOL
VAR_INPUT
END_VAR
Get_Done_Close:=closedone;
END_METHOD

METHOD Get_Done_Open : BOOL
VAR_INPUT
END_VAR
Get_Done_Open:=opendone;
END_METHOD

METHOD getErrID : UDINT
VAR_INPUT
	errID					:UDINT;//取值范围1~2
END_VAR
VAR
	nErrID					:UDINT;
END_VAR
nErrID:=errorID+errID;

getErrID:=nErrID;
END_METHOD

METHOD getErrTXT : STRING(255)
VAR_INPUT
	errID					:UDINT;//取值范围1~2
END_VAR
VAR
	sErrTXT					:STRING(255);
END_VAR

CASE errID OF
	1:
		sErrTXT:=CONCAT(STR1:=nameTXT,STR2:=' Open(TimeOut) Error!');
	2:
		sErrTXT:=CONCAT(STR1:=nameTXT,STR2:=' Close Error!');
	3:
		sErrTXT:=CONCAT(STR1:=nameTXT,STR2:=' NormalRun Error!');
	4:
		sErrTXT:=CONCAT(STR1:=nameTXT,STR2:=' CheckCondition Error!');
	5:
		sErrTXT:=CONCAT(STR1:=nameTXT,STR2:=' ParSet Fault!');
	6:
		sErrTXT:=CONCAT(STR1:=nameTXT,STR2:=' Communication Error!');
ELSE
	sErrTXT:=CONCAT(STR1:=nameTXT,STR2:='');
END_CASE
getErrTXT:=sErrTXT;
END_METHOD

METHOD getErrWTXT : WSTRING(255)
VAR_INPUT
	errID					:UDINT;//取值范围1~16
END_VAR
VAR
	sErrTXT					:WSTRING(255);
END_VAR

CASE errID OF
	1:
		sErrTXT:=WCONCAT(STR1:=TO_WSTRING(nameTXT),STR2:=" RF启动错误");
	2:
		sErrTXT:=WCONCAT(STR1:=TO_WSTRING(nameTXT),STR2:=" RF停止错误");
	3:
		sErrTXT:=WCONCAT(STR1:=TO_WSTRING(nameTXT),STR2:=" RF正常运行出现异常情况");
	4:
		sErrTXT:=WCONCAT(STR1:=TO_WSTRING(nameTXT),STR2:=" 检测到条件异常，关机处理");
	5:
		sErrTXT:=WCONCAT(STR1:=TO_WSTRING(nameTXT),STR2:=" 参数设置有误");
	6:
		sErrTXT:=WCONCAT(STR1:=TO_WSTRING(nameTXT),STR2:=" 通讯异常");
		
ELSE
	sErrTXT:=WCONCAT(STR1:=TO_WSTRING(nameTXT),STR2:="");
END_CASE
getErrWTXT:=sErrTXT;
END_METHOD

ACTION Init_ACT:
done:=(opendone OR closedone);
powerTon(IN:=mainPower,PT:=T#10S);
IF AlmAprSw AND powerTon.Q THEN
	errorStep:=5;
END_IF
IF readerror OR NOT readCondition AND firstPowerTON.Q THEN
	errorStep:=6;
END_IF
error:=error OR serialError OR NOT mainPower OR AlmAprSw;
InitHMI_ACT();
manualCtrl_ACT();
IF (error OR AlmAprSw OR ErrorAprSw OR NOT openCondition) AND openRelay THEN
	stop:=TRUE;
	busy:=FALSE;
	openRelay:=FALSE;
END_IF

noteTON_P(IN:=note_open,PT:=T#0.1S);
noteRTrig_P(CLK:=noteTON_P.Q);
IF noteRTrig_P.Q THEN
//	gLog_Note.append_EX(noteWTXT_Open);
END_IF
noteTON_N(IN:=note_close,PT:=T#0.1S);
noteRTrig_N(CLK:=noteTON_N.Q);
IF noteRTrig_N.Q THEN
//	gLog_Note.append_EX(noteWTXT_close);
END_IF
END_ACTION

ACTION InitHMI_ACT:
HMIItf.AlmAprSw:=AlmAprSw;
HMIItf.ErrorAprSw:=ErrorAprSw;

HMIItf.temperature:=temperature;
HMIItf.current:=current;
HMIItf.vol:=vol;

HMIItf.enableOpen:=enableOpenAprSw;
HMIItf.enableClose:=enableCloseAprSw;
HMIItf.HMIEnable:=hmiEN;
HMIItf.enable:=enable;
HMIItf.done:=done;
HMIItf.busy:=busy;
HMIItf.error:=error;
HMIItf.errID:=UDINT_TO_DINT(errID);
HMIItf.errTXT:=errTXT;
HMIItf.openRelay:=openRelay;
HMIItf.resetRelay:=resetRelay;

HMIItf.power:=power;
HMIItf.nameTXT:=nameTXT;

HMIItf.runTime:=runTime;
HMIItf.opencondition:=openCondition;
HMIItf.closecondition:=closeCondition;
END_ACTION

ACTION ManualCtrl_ACT:
//HMI手动控制
//IF ctrlMode=eManualCtrMode THEN
IF hmiEN THEN
	extendTrigRAlc(CLK:=HMIItf.extendAndretract);
	IF extendTrigRAlc.Q THEN// AND NOT busy
		IF openRelay THEN// 如果启动继电器或全速，则认为已经已启动完毕
			close:=TRUE;
		END_IF
		IF NOT openRelay THEN
			open:=TRUE;
		END_IF
	END_IF
	openendTrigR1_Aiko(CLK:=HMIItf.bopen);
	IF openendTrigR1_Aiko.Q AND NOT busy AND NOT openRelay THEN
		open:=TRUE;
		close:=FALSE;
	END_IF
	IF openendTrigR1_Aiko.Q AND busy AND openRelay THEN
		close:=TRUE;
		open:=FALSE;
	END_IF
	
	singleControltempR(CLK:=HMIItf.singleControltemp);
	openendTrigR1(CLK:=HMIItf.open);
	IF openendTrigR1.Q OR (singleControltempR.Q AND NOT openRelay ) THEN// AND NOT busy
		WarmHMI.showText:='';
		WarmHMI.showFlag:=TRUE;
		WarmHMI.showText:=CONCAT(WarmHMI.showText,'Are you sure you want to Open the ');
		WarmHMI.showText:=CONCAT(WarmHMI.showText,nameTXT);
		WarmHMI.showText:=CONCAT(WarmHMI.showText,' ?');
	END_IF
	IF WarmHMI.bOK AND NOT WarmHMI.showFlag AND FIND(WarmHMI.showText,nameTXT)>0 AND FIND(WarmHMI.showText,'Open')>0 THEN
		open:=TRUE;
		WarmHMI.bOK:=FALSE;
		WarmHMI.showText:='';
		operatorLog.append(CONCAT(CONCAT(nameTXT,' Open:'),UDINT_TO_STRING(setpower)));
		operatorLog.append(CONCAT(CONCAT(nameTXT,' Open:'),UDINT_TO_STRING(settime)));
	END_IF
	IF WarmHMI.bNO AND NOT WarmHMI.showFlag AND FIND(WarmHMI.showText,nameTXT)>0 AND FIND(WarmHMI.showText,'Open')>0 THEN
		WarmHMI.bNO:=FALSE;
		WarmHMI.showText:='';
	END_IF
	
	closeractTrigR1(CLK:=HMIItf.close);
	IF closeractTrigR1.Q OR (singleControltempR.Q AND openRelay) THEN// AND NOT busy
		WarmHMI.showText:='';
		WarmHMI.showFlag:=TRUE;
		WarmHMI.showText:=CONCAT(WarmHMI.showText,'Are you sure you want to Close the ');
		WarmHMI.showText:=CONCAT(WarmHMI.showText,nameTXT);
		WarmHMI.showText:=CONCAT(WarmHMI.showText,' ?');
	END_IF
	IF WarmHMI.bOK AND NOT WarmHMI.showFlag AND FIND(WarmHMI.showText,nameTXT)>0 AND FIND(WarmHMI.showText,'Close')>0 THEN
		close:=TRUE;
		operatorLog.append(CONCAT(nameTXT,' Close'));
		WarmHMI.bOK:=FALSE;
		WarmHMI.showText:='';
	END_IF
	IF WarmHMI.bNO AND NOT WarmHMI.showFlag AND FIND(WarmHMI.showText,nameTXT)>0 AND FIND(WarmHMI.showText,'Close')>0 THEN
		WarmHMI.bNO:=FALSE;
		WarmHMI.showText:='';
	END_IF
	
	resetTrigR1(CLK:=HMIItf.reset);
	IF resetTrigR1.Q THEN// AND NOT busy
		reset:=TRUE;
	END_IF
	
	stopTrigR1(CLK:=HMIItf.stop);
	IF stopTrigR1.Q THEN// AND NOT busy
		stop:=TRUE;
	END_IF
	
	powerTrigR1(CLK:=HMIItf.power);
	IF powerTrigR1.Q THEN// AND NOT busy
		IF power THEN
			power:=FALSE;
		ELSE
			power:=TRUE;
		END_IF
	END_IF
	
END_IF
END_ACTION

ACTION Open_ACT:
//分子泵伸出--open 触发
IF open AND NOT openCondition THEN
	note_open:=TRUE;
	note_close:=FALSE;
	NoteHMI.showFlag:=TRUE;
	NoteHMI.showText:='';
	NoteHMI.showText:=CONCAT(NoteHMI.showText,nameTXT);
	NoteHMI.showText:=CONCAT(NoteHMI.showText,' Open Condition Not Satisfied!');
	operatorLog.append(CONCAT(nameTXT,' Open Not Done '));
END_IF
IF open AND enable AND openCondition AND NOT AlmAprSw AND NOT ErrorAprSw AND NOT openbusy AND mainPower AND NOT resetRelay THEN// AND NOT busy
	note_open:=FALSE;
	note_close:=FALSE;
	busy:=TRUE;
	closebusy:=FALSE;
	openbusy:=TRUE;
	close:=FALSE;
	open:=FALSE;
	done:=FALSE;
	opendone:=FALSE;
	closedone:=FALSE;
	openStep:=10;
	writeStep:=0;
	writeMaxStep:=0;
	readAndWriteLock:=TRUE;
	// searial_send(setPoint)**************************************
	closeStep:=0;
	operatorLog.append(CONCAT(nameTXT,' Open Done '));
END_IF
open:=FALSE;
runTimeClearR(CLK:=HMIItf.runTimeClear);
runTON(IN:=NOT error AND openRelay AND NOT runTON.Q, PT:=T#60S);// 1小时计数一次,启动，无报错，且全速
IF runTON.Q AND runTime<999999999999999 AND NOT runTimeClearR.Q THEN
	runTime:=runTime+1;
END_IF
IF runTimeClearR.Q THEN
	runTime:=0;
END_IF
//IF NOT openRelay AND NOT AccAprSw AND NOT DccAprSw AND NOT NormalAprSw THEN// 计数清零
//	runTime:=0;
//END_IF

CASE openStep OF
0:
	//ready
	runTON(IN:=FALSE);
	openErrorDelayTon(IN:=FALSE);
	openErrorDelayTon(IN:=FALSE);
	openDoneDelayTon(IN:=FALSE);
	t1(IN:=FALSE);
	rematime:=0;
10:
	IF setpower<1 OR (NOT co_control AND settime<1) THEN 
		open:=FALSE;
		close:=FALSE;
		openbusy:=FALSE;
		closebusy:=FALSE;
		errorStep:=5;
		openStep:=60;
	ELSE
		t1(IN:=readStep<10 AND writeStep<10 AND writeMaxStep<10,PT:=T#0.5S);
		IF t1.Q THEN
			openErrorDelayTon(IN:=FALSE);
			openDoneDelayTon(IN:=FALSE);
			openStep:=15;
			openRelay:=TRUE;
			setpointdone:=FALSE;
			Act_Write_1();
			openbusy:=TRUE;
			closebusy:=FALSE;
			closeRelay:=FALSE;
			t1(IN:=FALSE);
		END_IF
	END_IF
15:
	t1(IN:=setpointdone,PT:=T#0.1S);
	IF t1.Q THEN
		setpointdone:=FALSE;
		t1(IN:=FALSE);
		PLC_PowerRF.receiveFlag:=FALSE;
		PLC_PowerRF.WriteStart();
		openStep:=17;
	END_IF
17:
	t1(IN:=PLC_PowerRF.receiveFlag,PT:=T#0.05S);
	IF t1.Q THEN
		t1(IN:=FALSE);
		PLC_PowerRF.receiveFlag:=FALSE;
		readAndWriteLock:=FALSE;
		busy:=false;
		openStep:=20;
	END_IF
20:
	// AccAprSw可以看成是forward Power > 5 ,< set point - 5// 或者反射功率>0
	openErrorDelayTon(IN:=(NOT (ABS(forwardpower)>=0 AND reflectedpower<10 AND ABS(setpower-forwardpower)<2)),PT:=errorDelayTime);
	IF openErrorDelayTon.Q THEN
		//done:=FALSE;
		open:=FALSE;
		close:=FALSE;
		openbusy:=FALSE;
		closebusy:=FALSE;
		errorStep:=1;
		openStep:=60;
		RETURN;
	END_IF
	IF enableopenAprSw THEN
		openDoneDelayTon(IN:=ABS(forwardpower)>=0 AND reflectedpower<10 AND ABS(setpower-forwardpower)<2,PT:=doneDelayTimeShortopenend);
	END_IF
	IF openDoneDelayTon.Q THEN
		openErrorDelayTon(IN:=FALSE);
		openDoneDelayTon(IN:=FALSE);
		openStep:=30;
	END_IF
	
	//状态实时检测
	IF NOT openCondition AND (NOT closedone OR openRelay) THEN// 检测到开条件消失，强制关闭
		openRelay:=FALSE;
		errorStep:=4;
		openbusy:=FALSE;
		closebusy:=FALSE;
		openStep:=60;
	END_IF
	IF (ErrorAprSw OR AlmAprSw) AND openRelay THEN//只要报错；启动线圈启动，强锁启动信号
		openRelay:=FALSE;
		openStep:=60;/////
		errorStep:=3;
		openbusy:=FALSE;
		closebusy:=FALSE;
	END_IF
30:
	openErrorDelayTon(IN:=NOT co_control,PT:=UDINT_TO_TIME(settime*1000));// 反射调整超时时间
	rematime:=TIME_TO_UDINT(openErrorDelayTon.ET/1000);
	rematime:=settime-rematime;
	IF openErrorDelayTon.Q OR co_control THEN
		openStep:=40;
		rematime:=0;
		openErrorDelayTon(IN:=FALSE);
	END_IF
	// 状态实时检测
	IF NOT openCondition AND (NOT closedone OR openRelay) THEN//蝶阀单控，检测到开条件消失，强制关闭
		openRelay:=FALSE;
		errorStep:=4;
		openStep:=60;
		closebusy:=FALSE;
		openbusy:=FALSE;
	END_IF
	IF (ErrorAprSw OR AlmAprSw) AND openRelay THEN//只要报错；启动线圈启动，强锁启动信号
		openRelay:=FALSE;
		stop:=TRUE;
		openStep:=60;/////
		errorStep:=3;
		closebusy:=FALSE;
		openbusy:=FALSE;
	END_IF
40:
	busy:=FALSE;
	IF NOT co_control THEN
		openRelay:=FALSE;
		close:=TRUE;
	END_IF
	openStep:=50;
	openbusy:=FALSE;
	readAndWriteLock:=FALSE;
	opendone:=TRUE;
50:
	rematime:=0;
60:
	openRelay:=FALSE;
	openStep:=70;
	busy:=FALSE;
	readAndWriteLock:=FALSE;
	;//报错
	co_control:=FALSE;
	opendone:=FALSE;
END_CASE
END_ACTION

ACTION Read_ACT:
//气缸收回--read 触发
firstPowerTON(IN:=firstPower,PT:=T#10S);
readTON(IN:=NOT readAndWriteLock AND NOT busy AND  NOT readbusy AND readStep=0 AND readCondition,PT:=T#0.05S);
IF readTON.Q THEN// AND NOT busy
	readdone:=FALSE;
	readStep:=10;
	readbusy:=TRUE;
	readerror:=FALSE;
END_IF
CASE readStep OF
0:
	//ready
	readTon1(IN:=FALSE);
	readTon2(IN:=FALSE);
	readTon3(IN:=FALSE);
10:// State
	IF gICP.PowerRF.controlMode=2 THEN
		PLC_PowerRF.readStateFlag:=FALSE;
		PLC_PowerRF.ReadState();
		readStep:=readStep+10;
	ELSE
		PLC_PowerRF.readStateFlag:=FALSE;
		PLC_PowerRF.WriteRS232Mode();
		readStep:=readStep+15;
		PLC_PowerRF.receiveFlag:=FALSE;
	END_IF
20:
	IF PLC_PowerRF.readStateFlag THEN
		PLC_PowerRF.readStateFlag:=FALSE;
		// 数据处理
		readTon1(IN:=FALSE);
		readStep:=readStep+10;
		RETURN;
	END_IF
	readTon1(IN:=TRUE,PT:=T#500MS);// 超时
	IF readTon1.Q THEN
		readStep:=6000;
		readTon1(IN:=FALSE);
		readTon2(IN:=FALSE);
		RETURN;
	END_IF
25:
	IF PLC_PowerRF.receiveFlag THEN
		PLC_PowerRF.receiveFlag:=FALSE;
		// 数据处理
		readTon1(IN:=FALSE);
		readStep:=readStep+5;
		RETURN;
	END_IF
	readTon1(IN:=TRUE,PT:=T#500MS);// 超时
	IF readTon1.Q THEN
		readStep:=6000;
		readTon1(IN:=FALSE);
		readTon2(IN:=FALSE);
		RETURN;
	END_IF
30:
	readTon3(IN:=TRUE,PT:=T#0.1S);
	IF readTon3.Q THEN
		readStep:=readStep+10;
		readTon3(IN:=FALSE);
	END_IF
40:// State
	PLC_PowerRF.readStateFlag:=FALSE;
	PLC_PowerRF.ReadState();
	readStep:=readStep+10;
50:
	IF PLC_PowerRF.readStateFlag THEN
		PLC_PowerRF.readStateFlag:=FALSE;
		// 数据处理
		readTon1(IN:=FALSE);
		readStep:=readStep+10;
		RETURN;
	END_IF
	readTon1(IN:=TRUE,PT:=T#500MS);// 超时
	IF readTon1.Q THEN
		readStep:=6000;
		readTon1(IN:=FALSE);
		readTon2(IN:=FALSE);
		RETURN;
	END_IF
60:
	readStep:=90;
90:
	readTon3(IN:=TRUE,PT:=T#0.1S);
	IF readTon3.Q THEN
		readStep:=5000;
		readTon3(IN:=FALSE);
	END_IF
5000:
	readbusy:=FALSE;
	readdone:=TRUE;
	readStep:=0;
	readerror:=FALSE;
	PLC_PowerRF.ClearCom:=TRUE;
6000:
	readbusy:=FALSE;
	readdone:=TRUE;
	readStep:=0;
	readErrorTimes:=readErrorTimes+1;
	IF readErrorTimes>3 THEN
		readErrorTimes:=0;
		readerror:=TRUE;
		gICP.PowerRF.setpowerRead:=0;
		gICP.PowerRF.forwardpower:=0;
		gICP.PowerRF.reflectedpower:=0;
		gICP.PowerRF.maxpower:=0;
	END_IF
	gICP.PowerRF.controlMode:=0;
END_CASE
END_ACTION

ACTION Reset_ACT:
IF reset THEN
	IF NOT power THEN
		openRelay:=FALSE;
		closeRelay:=FALSE;
	END_IF
	note_open:=FALSE;
	note_close:=FALSE;
	IF errorStep<>0 OR  AlmAprSw OR ErrorAprSw THEN
		errorStep:=0;
		busy:=FALSE;
		closebusy:=FALSE;
		openbusy:=FALSE;
		resetRelay:=TRUE;
		readAndWriteLock:=TRUE;
		PLC_PowerRF.WriteReset();
	END_IF
	reset:=FALSE;
	note_open:=FALSE;
	note_close:=FALSE;
END_IF
resetRelayTON(IN:=resetRelay , PT:=resetRelayTONTime);
IF resetRelayTON.Q THEN
	errorStep:=0;
	busy:=FALSE;
	resetRelay:=FALSE;
	readAndWriteLock:=FALSE;
END_IF

IF stop THEN
	note_open:=FALSE;
	note_close:=FALSE;
	stop:=FALSE;
	openRelay:=FALSE;
	closeRelay:=FALSE;
	//无自锁检测说法，直接停
	openStep:=0;
	closeStep:=0;
	writeStep:=0;
	writeMaxStep:=0;
END_IF
END_ACTION

ACTION VersionLog:
(*
版本: V1.0.0.0
说明:
	1. 首个版本
	2. 含普通分子泵\泵组类型的控制
	3. 可配置是否有到位信号, 以及到位稳定时间
(--------------------------------------------------)
新版本: V1.0.1.0
更新时间: 2019/11/20 19:00
更新说明:
	1. 优化编写方式
	2. 修改错误编码起始位，现改为从1开始
(--------------------------------------------------)
新版本: V1.0.1.1
更新时间: 2020/03/23 23:00
更新说明:
	1. 优化报错方式
	2. 增加伸出、缩回、复位和停止触发函数
(--------------------------------------------------)
新版本: V1.0.1.2
更新时间: 2020/04/22 09:50
更新说明:
	1. 增加中文报警输出
(--------------------------------------------------)
新版本: V1.0.1.3
更新时间: 2020/09/16
更新说明:
	1. 开放错误ID、错误文本信息获取接口
(--------------------------------------------------)
新版本: V1.0.1.4
更新时间: 2020/10/06
更新说明:
	1. 移除控制模式变量，增加HMI启用条件
	2. 增加外部获取伸出缩回完成信号接口函数
(--------------------------------------------------)
新版本: V1.0.1.5
更新时间: 2020/10/14
更新说明:
	1. 优化代码
(--------------------------------------------------)
新版本: V2.0.1.0
更新时间: 2023/11/17
更新说明:
	1. 分子泵控制独立
(--------------------------------------------------)


*)
END_ACTION

ACTION WriteMaxPower_ACT:
//分子泵--writeMax 触发

CASE writeMaxStep OF
0:
	//ready
	writeMaxTON(IN:=FALSE);
10:
	writeMaxTON(IN:=readStep<10,PT:=T#0.1S);
	IF writeMaxTON.Q THEN
		PLC_PowerRF.ClearCom:=TRUE;
		writeMaxTON(IN:=FALSE);
		writeMaxStep:=writeMaxStep+10;
	END_IF
20:
	IF readStep<10 AND openStep<10 AND closeStep<10 AND writeMaxStep<10 THEN
		PLC_PowerRF.WriteMaxPower(gICP.PowerRF.setpower);
		PLC_PowerRF.receiveFlag:=FALSE;
		writeMaxStep:=writeMaxStep+10;
	END_IF
30:
	writeMaxTON(IN:=NOT PLC_PowerRF.receiveFlag ,PT:=T#0.5S);
	IF writeMaxTON.Q THEN
		PLC_PowerRF.receiveFlag:=FALSE;
		writeMaxTON(IN:=FALSE);
		writeMaxStep:=writeMaxStep+10;
		RETURN;
	END_IF
	IF PLC_PowerRF.receiveFlag THEN
		PLC_PowerRF.receiveFlag:=FALSE;
		writeMaxTON(IN:=FALSE);
		writeMaxStep:=writeMaxStep+10;
		RETURN;
	END_IF
40:
	writeMaxStep:=100;
100:
	writeMaxStep:=0;	
	readAndWriteLock:=FALSE;
END_CASE
END_ACTION

ACTION WritePower_ACT:
//分子泵--write 触发

CASE writeStep OF
0:
	//ready
	writeTON(IN:=FALSE);
10:
	writeTON(IN:=readStep<10,PT:=T#0.1S);
	setpointdone:=FALSE;
	IF writeTON.Q THEN
		PLC_PowerRF.ClearCom:=TRUE;
		writeTON(IN:=FALSE);
		writeStep:=writeStep+10;
	END_IF
20:
	IF readStep<10  AND writeMaxStep<10 THEN
		PLC_PowerRF.WritePower(gICP.PowerRF.setpower);
		PLC_PowerRF.receiveFlag:=FALSE;
		writeStep:=writeStep+10;
	END_IF
30:
	writeTON(IN:=NOT PLC_PowerRF.receiveFlag ,PT:=T#0.5S);
	IF writeTON.Q THEN
		PLC_PowerRF.receiveFlag:=FALSE;
		writeTON(IN:=FALSE);
		writeStep:=writeStep+10;
		setpointdone:=FALSE;
		RETURN;
	END_IF
	IF PLC_PowerRF.receiveFlag THEN
		PLC_PowerRF.receiveFlag:=FALSE;
		writeTON(IN:=FALSE);
		writeStep:=writeStep+10;
		setpointdone:=TRUE;
		RETURN;
	END_IF
40:
	writeStep:=100;
100:
	writeStep:=0;	
	readAndWriteLock:=FALSE;
END_CASE
END_ACTION

END_FUNCTION_BLOCK

// ---- POUs/Communication/PLC_PowerRF.TcPOU
PROGRAM PLC_PowerRF
VAR_INPUT
	nSocketType:UINT:=0;// socket 类型; 0 表示 server; 1 表示 client;
	sTerminalName:STRING;// 通讯对方名称 自定义
	sHost:STRING(20):='127.0.0.1';// 通讯IP地址; server时表示本地host; client时表示远程host
	nPort:UDINT:=8900;// 通讯端口号;
	bEnable:BOOL:=TRUE;// 通讯启用\禁用连接
	sSendSuffix:STRING:='';//此处可统一添加发送后缀字符 $R$N
	nQueueInterval:UDINT:=50;// 发送队列时间间隔 单位ms
	logHandleArray:ARRAY [1..5] OF POINTER TO printLogModule_EX;// log 操作 handle 数组
	logHandleArrayLength:UINT:=0;// log 操作 handle 数组长度, 不超过5
	readStateFlag:BOOL;
	ClearCom:BOOL;
	receiveFlag:BOOL;
END_VAR
VAR_OUTPUT
	bSendCondition	:BOOL;//可发送条件
	bSocketConnected:BOOL;//连接状态
END_VAR
VAR CONSTANT
	cNumBegin		:DINT:=1;
	cNumEnd			:DINT:=100;
END_VAR
VAR
	sendDataArray	:ARRAY [cNumBegin..cNumEnd] OF STRING(255);
	length			:DINT:=0;
	endPoint		:DINT:=cNumBegin;
	popupSendData	:STRING(255);
	//popup
	popupStep		:UINT:=0;
	popupTON1		:TON;
	popupTON2		:TON;
	iPopup			:DINT:=0;
	_PopupLength	:DINT:=0;
END_VAR
VAR
	tcpipClient					:tcpipClientModule_EX;
	tcpipServer					:tcpipServerModule_EX;////定义服务器对象
	
	tcpipSendDataBuff_Server	:STRING(255);//发送数据 Buff server
	tcpipSendDataBuff_Client	:STRING(255);//发送数据 Buff client
	
	tcpipSendDataClear			:STRING(255);//发送数据 清空
	tcpipSendData				:STRING(255);//发送数据
	
	tcpipRecDataBuff_Server		:STRING(255);//已接收数据 Buff server
	tcpipRecDataBuff_Client		:STRING(255);//已接收数据 Buff client
	
	tcpipRecDataClear			:STRING(255);//已接收数据 清空
	tcpipRecData				:STRING(255);//已接收数据
	
	tcpConnectR_Trig			:R_Trig;//初始连接上升沿
	tcpConnectF_Trig			:F_Trig;//初始连接下降沿
	registerStep				:UDINT;//ALC注册控制步
	registerTON					:TON;//ALC注册延时
	
	logHandleArray_index		:UINT:=1;
END_VAR
VAR
	bTrig_Start:BOOL;
	rTrig_Start:R_TRIG;
	tTrig_Start:TON;
	
	bTrig_Stop:BOOL;
	rTrig_Stop:R_TRIG;
	tTrig_Stop:TON;
	
	bTrig_Reset:BOOL;
	rTrig_Reset:R_TRIG;
	tTrig_Reset:TON;
	
	
	bTrig_Init:BOOL;
	rTrig_Init:R_TRIG;
	
	bTrig_All_Home:BOOL;
	rTrig_All_Home:R_TRIG;
	
	bTrig_Z_Safe:BOOL;
	rTrig_Z_Safe:R_TRIG;
	
	bTrig_P_Pos_:BOOL;
	rTrig_P_Pos_:R_TRIG;
	nTrig_P_Pos_TrayNum:UINT:=1;
	nTrig_P_Pos_RowNum:UINT:=1;
	
	bTrig_Move_P_:BOOL;
	rTrig_Move_P_:R_TRIG;
	nTrig_Move_P_TrayNum:UINT:=1;
	nTrig_Move_P_RowNum:UINT:=1;
	nTrig_Move_P_PosNum:UINT:=1;
	findposstart	:INT;
	findposend		:INT;
	find_pos		:INT;
	recStrTemp		:STRING(255);
END_VAR


CASE nSocketType OF
0://TCPIP server
	tcpipServer(
		sSrvNetId:= , 
		sLocalHost:=sHost , 
		nLocalPort:=nPort , 
		bStartConnect:=bEnable , 
		tcpipSDataLen:=TO_UDINT(LEN(tcpipSendDataBuff_Server)) , 
		tcpipSData:=ADR(tcpipSendDataBuff_Server) , 
		bSend:= , 
		tcpipRecDataLen:=SIZEOF(tcpipRecDataBuff_Server) , 
		tcpipRecData:=ADR(tcpipRecDataBuff_Server) , 
		bAccepted=> , 
		bSendBusy=> , 
		bRecData=> );
	bSendCondition:=tcpipServer.bAccepted AND NOT tcpipServer.bSendBusy;
	//TCPIP连接
	bSocketConnected:=tcpipServer.bAccepted;
	IF NOT tcpipServer.bAccepted THEN
		length:=0;
		endPoint:=cNumBegin;
	END_IF
	tcpConnectR_Trig(CLK:=tcpipServer.bAccepted);
	tcpConnectF_Trig(CLK:=tcpipServer.bAccepted);

1://TCPIP client
	tcpipClient(
		sSrvNetId:= , 
		sRemoteHost:=sHost , 
		nRemotePort:=nPort , 
		bStartConnect:=bEnable , 
		tcpipSDataLen:=TO_UDINT(LEN(tcpipSendDataBuff_Client)) , 
		tcpipSData:=ADR(tcpipSendDataBuff_Client) , 
		bSend:= , 
		tcpipRecDataLen:=SIZEOF(tcpipRecDataBuff_Client) , 
		tcpipRecData:=ADR(tcpipRecDataBuff_Client) , 
		bConnected=> , 
		bSendBusy=> , 
		bRecData=> );
	bSendCondition:=tcpipClient.bConnected AND NOT tcpipClient.bSendBusy;
	//TCPIP连接
	bSocketConnected:=tcpipClient.bConnected;
	IF NOT tcpipClient.bConnected THEN
		length:=0;
		endPoint:=cNumBegin;
	END_IF
	tcpConnectR_Trig(CLK:=tcpipClient.bConnected);
	tcpConnectF_Trig(CLK:=tcpipClient.bConnected);
END_CASE
IF ClearCom THEN
	length:=0;
	endPoint:=cNumBegin;
	ClearCom:=FALSE;
END_IF
IF tcpConnectR_Trig.Q THEN
	FOR logHandleArray_index:=1 TO logHandleArrayLength DO
		logHandleArray[logHandleArray_index]^.append(CONCAT(sTerminalName, ' has been connected'));
	END_FOR
	registerStep:=10;
END_IF
IF tcpConnectF_Trig.Q THEN
	FOR logHandleArray_index:=1 TO logHandleArrayLength DO
		logHandleArray[logHandleArray_index]^.append(CONCAT(sTerminalName, ' has been disconnected'));
	END_FOR
	registerStep:=0;
END_IF
//数据接收处理
CASE nSocketType OF
0://TCPIP server
	IF tcpipServer.bRecData THEN
		tcpipRecData:=tcpipRecDataBuff_Server;//buff转存
		tcpipRecDataBuff_Server:=tcpipRecDataClear;//转存之后清空buff
		dataProcessing();
	END_IF
1://TCPIP client
	IF tcpipClient.bRecData THEN
		tcpipRecData:=tcpipRecDataBuff_Client;//buff转存
		tcpipRecDataBuff_Client:=tcpipRecDataClear;//转存之后清空buff
		dataProcessing();
	END_IF
END_CASE


popup();

CASE registerStep OF
0:
	//Ready
END_CASE

METHOD appendSend : BOOL
VAR_INPUT
	str			:STRING(255);
END_VAR
VAR
	suffix					:STRING;
	strTemp_appendSend		:STRING(255);
END_VAR

IF endPoint>(cNumEnd-1) THEN
	RETURN;
END_IF
suffix:=sSendSuffix;//此处可统一添加发送后缀字符 $R$N

strTemp_appendSend:=CONCAT(str,suffix);
sendDataArray[endPoint]:=strTemp_appendSend;

endPoint:=endPoint+1;
length:=endPoint-cNumBegin;
END_METHOD

METHOD dataProcessing : BOOL
VAR_INPUT
END_VAR
VAR
	strTemp:STRING;
END_VAR
FOR logHandleArray_index:=1 TO logHandleArrayLength DO
	CASE nSocketType OF
	0://TCPIP server
//		logHandleArray[logHandleArray_index]^.append(CONCAT(CONCAT(CONCAT('Recevie From ', sTerminalName), ' -- '),tcpipRecData));
	1://TCPIP client
//		logHandleArray[logHandleArray_index]^.append(CONCAT(CONCAT(CONCAT('Recevie From ', sTerminalName), ' -- '),tcpipRecData));
	END_CASE
END_FOR
receiveFlag:=TRUE;
findposend:=0;
find_pos:=0;
IF MID(tcpipRecData,1,32)='$R' AND MID(tcpipRecData,1,33)='$R'  THEN
	gICP.PowerRF.controlMode:=STRING_TO_INT(MID(tcpipRecData,1,1));
	gICP.PowerRF.outputMode:=STRING_TO_INT(MID(tcpipRecData,1,2));
	gICP.PowerRF.outputState:=STRING_TO_INT(MID(tcpipRecData,1,3));
	strTemp:='';
	strTemp:=CONCAT(strTemp,(MID(tcpipRecData,2,6)));
	gICP.PowerRF.alarmState:=STRING_TO_INT(strTemp);
	strTemp:='';
	strTemp:=CONCAT(strTemp,(MID(tcpipRecData,5,9)));
	gICP.PowerRF.setpowerRead:=STRING_TO_UDINT(strTemp);
	strTemp:='';
	strTemp:=CONCAT(strTemp,(MID(tcpipRecData,5,15)));
	gICP.PowerRF.forwardpower:=STRING_TO_UDINT(strTemp);
	strTemp:='';
	strTemp:=CONCAT(strTemp,(MID(tcpipRecData,5,21)));
	gICP.PowerRF.reflectedpower:=STRING_TO_UDINT(strTemp);
	strTemp:='';
	strTemp:=CONCAT(strTemp,(MID(tcpipRecData,5,27)));
	gICP.PowerRF.maxpower:=STRING_TO_UDINT(strTemp);
	readStateFlag:=TRUE;
END_IF
END_METHOD

METHOD PRIVATE popup : BOOL
VAR_INPUT
END_VAR
CASE popupStep OF
0:
	IF length>0 AND bSendCondition THEN
		_PopupLength:=length;
		popupSendData:=sendDataArray[cNumBegin];
		FOR iPopup:=cNumBegin TO (_PopupLength-1) DO
			sendDataArray[iPopup]:=sendDataArray[iPopup+1];
		END_FOR
		endPoint:=endPoint-1;
		length:=endPoint-cNumBegin;
		sendData(popupSendData);//此处是调用信息发送
		popupStep:=10;
	END_IF
10:
	popupTON2(IN:=NOT popupTON2.Q, PT:=T#2S);
	IF NOT bSendCondition OR popupTON2.Q THEN
		popupTON2(IN:=FALSE);
		popupStep:=11;
	END_IF
11:
	IF bSendCondition THEN
		popupStep:=12;
	END_IF
	popupTON1(IN:=FALSE);
12:
	//popupTON1(IN:=NOT popupTON1.Q,PT:=T#10MS);
	popupTON1(IN:=NOT popupTON1.Q,PT:=TO_TIME(nQueueInterval));
	IF popupTON1.Q THEN
		popupStep:=0;
	END_IF
END_CASE
END_METHOD

METHOD ReadState : BOOL
VAR_INPUT
END_VAR
VAR
END_VAR
appendSend('Q$R');
END_METHOD

METHOD PRIVATE sendData : BOOL
VAR_INPUT
	dataStruct	:STRING(255);
END_VAR
IF bSendCondition AND bEnable THEN
	tcpipSendData:=dataStruct;
	
	CASE nSocketType OF
	0://TCPIP server
		tcpipSendDataBuff_Server:=tcpipSendData;
		tcpipSendData:=tcpipSendDataClear;	
		tcpipServer.bSend:=TRUE;
	1://TCPIP client
		tcpipSendDataBuff_Client:=tcpipSendData;
		tcpipSendData:=tcpipSendDataClear;	
		tcpipClient.bSend:=TRUE;
	END_CASE
	
	FOR logHandleArray_index:=1 TO logHandleArrayLength DO
		CASE nSocketType OF
		0://TCPIP server
//			logHandleArray[logHandleArray_index]^.append(CONCAT(CONCAT(CONCAT('Send To ', sTerminalName), ' -- '),tcpipSendDataBuff_Server));
		1://TCPIP client
//			logHandleArray[logHandleArray_index]^.append(CONCAT(CONCAT(CONCAT('Send To ', sTerminalName), ' -- '),tcpipSendDataBuff_Client));
		END_CASE
	END_FOR
END_IF
END_METHOD

METHOD WriteMaxPower : BOOL
VAR_INPUT
	maxpowerpoint:UDINT;
END_VAR
VAR
	str:STRING;
	_bit:UDINT;
	_ten:UDINT;
	_hundred:UDINT;
	_thousand:UDINT;
END_VAR
str:='';
_thousand:=maxpowerpoint/1000;
str:=CONCAT(str,UDINT_TO_STRING(maxpowerpoint));
//_hundred:=maxpowerpoint/100 MOD 10;
//str:=CONCAT(str,UDINT_TO_STRING(_hundred));
//_ten:=maxpowerpoint/10 MOD 10;
//str:=CONCAT(str,UDINT_TO_STRING(_ten));
//_bit:=maxpowerpoint MOD 10;
//str:=CONCAT(str,UDINT_TO_STRING(_bit));
str:=CONCAT(str,' M$R');
appendSend(str);
END_METHOD

METHOD WritePower : BOOL
VAR_INPUT
	powerpoint:UDINT;
END_VAR
VAR
	str:STRING;
	_bit:UDINT;
	_ten:UDINT;
	_hundred:UDINT;
	_thousand:UDINT;
END_VAR
str:='';
//_thousand:=powerpoint/1000;
str:=CONCAT(str,UDINT_TO_STRING(powerpoint));
//_hundred:=powerpoint/100 MOD 10;
//str:=CONCAT(str,UDINT_TO_STRING(_hundred));
//_ten:=powerpoint/10 MOD 10;
//str:=CONCAT(str,UDINT_TO_STRING(_ten));
//_bit:=powerpoint MOD 10;
//str:=CONCAT(str,UDINT_TO_STRING(_bit));
str:=CONCAT(str,' W$R');
appendSend(str);
END_METHOD

METHOD WriteReset : BOOL
VAR_INPUT
		

END_VAR
appendSend('RESET$R');
END_METHOD

METHOD WriteRS232Mode : BOOL
VAR_INPUT
		

END_VAR
appendSend('***$R');
END_METHOD

METHOD WriteStart : BOOL
VAR_INPUT
		

END_VAR
appendSend('G$R');
END_METHOD

METHOD WriteStop : BOOL
VAR_INPUT
		

END_VAR
appendSend('S$R');
END_METHOD

END_PROGRAM

// ---- POUs/BaseModule/ActionModule/chillerModule/ChillerModule_1.TcPOU
(*
--报错编号0: 无报错
--报错编号1: Extend Error
--报错编号2: Retract Error
*)
FUNCTION_BLOCK ChillerModule_1
VAR_IN_OUT
	WarmHMI					:WARMStruct;
	NoteHMI					:NoteStruct;
	operatorLog				:printLogModule_EX;
END_VAR
VAR_INPUT
	HMIItf						:ChillerModuleHMI;//每个Chiller对象都关联了一个HMI
	ChillerType				:ChillerType:=ChillerType_Default;//设置Chiller的类型, 可通过该变量修改为真空发生器
	
	real_TimeMonitor			:BOOL:=TRUE;//实时状态检测
	
	extend						:BOOL:=FALSE;//伸出触发信号
	extCondition				:BOOL:=TRUE;//伸出启停条件
	retract						:BOOL:=FALSE;//收回触发信号
	retCondition				:BOOL:=TRUE;//收回启停条件
	setPoint					:BOOL:=FALSE;//设置触发信号
	setCondition				:BOOL:=TRUE;//设置启停条件
	readPoint					:BOOL:=FALSE;// 设置读取信号
	readCondition				:BOOL:=TRUE;// 设置读取条件
	reset						:BOOL:=FALSE;//复位信号
	stop						:BOOL:=FALSE;//停止信号
	power						:BOOL:=TRUE;//Chiller动作后是否关闭继电器得电状态, TRUE--保持得电,FALSE--断开得电
	enable						:BOOL:=TRUE;//Chiller禁用条件
	//ctrlMode					:ControlMode:=ControlMode.eManualCtrMode;//eManualCtrMode or eAutoCtrMode
	hmiEN						:BOOL:=TRUE;//HMI 启用条件
	
	errorDelayTime				:TIME:=T#3000MS;//Chiller感应器感应超时
	//doneDelayTimeShort		:TIME:=T#100MS;//Chiller感应到位延时---取消使用
	//doneDelayTimeLong			:TIME:=T#500MS;//无Chiller感应到位延时---取消使用
	doneDelayTimeShortExtend	:TIME:=T#100MS;//Chiller感应到位延时_伸出
	doneDelayTimeShortRetract	:TIME:=T#100MS;//Chiller感应到位延时_收回
	doneDelayTimeLongExtend		:TIME:=T#500MS;//无Chiller感应到位延时_伸出
	doneDelayTimeLongRetract	:TIME:=T#500MS;//无Chiller感应到位延时_收回
	doneDelayTimeLongSET		:TIME:=T#500MS;//无Chiller感应到位延时_SET
	errorID						:UDINT:=0;//Chiller错误报警分配的起始ID
	nameTXT						:STRING(255):='';//Chiller名字
	
	extAprSw					:BOOL:=FALSE;//Chiller伸出感应器信号,需要链接到实际的IO点
	retAprSw					:BOOL:=FALSE;//Chiller收回感应器信号,需要链接到实际的IO点
	enableExtAprSw				:BOOL:=TRUE;//启用伸出感应器,针对只有一个传感器的Chiller
	enableRetAprSw				:BOOL:=TRUE;//启用收回感应器,针对只有一个传感器的Chiller
	
	noteWTXT_Ext				:WSTRING(255):="";//Chiller伸出动作NoteTXT 中文
	noteWTXT_Ret				:WSTRING(255):="";//Chiller缩回动作NoteTXT 中文
	pumon:BOOL;		
	uinton:BOOL;
	fault:BOOL;
	unitstoping:BOOL;
	alarmTemperatureH			:REAL:=30;
	alarmTemperatureL			:REAL:=10;
	RTD1:REAL;
	RTD2:REAL;
	setpointVal					:REAL;
END_VAR
VAR_OUTPUT
	extRelay				:BOOL:=FALSE;//Chiller伸出执行继电器,需要链接到实际的IO点
	retRelay				:BOOL:=FALSE;//Chiller收回执行继电器,需要链接到实际的IO点
	note_Ext				:BOOL:=FALSE;// 操作提示：true 伸出、打开执行无法下发
	note_Ret				:BOOL:=FALSE;// 操作提示：true 缩回、关闭执行无法下发
	note_Set				:BOOL:=FALSE;// 操作提示：true 设置参数执行无法下发
	busy					:BOOL;//Chiller动作Busy状态
	readbusy				:BOOL;
	readerror				:BOOL;
	done					:BOOL;//Chiller动作Done状态
	extdone					:BOOL;//Chiller动作伸出完成
	retdone					:BOOL;//Chiller动作收回完成
	setdone					:BOOL;//Chiller动作收回完成
	readdone				:BOOL;//Chiller动作收回完成
	error					:BOOL;//Chiller动作error状态
	errID					:UDINT;//Chiller动作errID
	errTXT					:STRING(255):='';//Chiller动作errTXT
	errWTXT					:WSTRING(255):="";//Chiller动作errTXT 中文
	sensorShow				:STRING;
END_VAR
	
VAR
	readAndWriteLock:BOOL;
	firstPower:BOOL:=TRUE;
	extErrorDelayTon		:Ton;
	extDoneDelayTon			:Ton;
	retErrorDelayTon		:Ton;
	retDoneDelayTon			:Ton;
	setErrorDelayTon		:Ton;
	setDoneDelayTon			:Ton;
	readConditionTon		:TON;
	readTon1				:TON;
	readTon2				:TON;
	
	extendTrigRAlc			:R_Trig;//上升沿触发
	
	singleControlR			:R_Trig;//上升沿触发
	singleControlF			:F_Trig;//上升沿触发
	
	setR					:R_Trig;//上升沿触发
	
	extendTrigR1			:R_Trig;//上升沿触发
	retractTrigR1			:R_Trig;//上升沿触发
	resetTrigR1				:R_Trig;//上升沿触发
	stopTrigR1				:R_Trig;//上升沿触发
	powerTrigR1				:R_Trig;//上升沿触发
	
	extStep					:UINT:=0;
	retStep					:UINT:=0;
	setStep					:UINT:=0;
	readStep				:UINT:=0;
	errorStep				:UINT:=0;
	
	notBusyMonitorDelayTon:TON;//动作不切换时，延迟检测
	notBusyMonitorDelayTime:TIME:=T#2S;//动作不切换延迟检测时间
	noteTON_P:tON;            // 操作提示标志位延时继电器
	noteTON_N:tON;            // 操作提示标志位延时继电器
	noteRTrig_P:R_TRIG;          // 操作提示
	noteRTrig_N:R_TRIG;          // 操作提示
	extRealayRtrig:R_TRIG;
	retRealayRtrig:R_TRIG;
END_VAR

// 实时读取设置的流量值以及实际反馈浏览值
// ****************************
Init_ACT();
Error_ACT();
Extend_ACT();
Retract_ACT();
Reset_ACT();
Set_ACT();
Read_ACT();
Error_ACT();
SafeMonitor_ACT();

(*
触发伸出动作，成功触发返回TRUE，触发失败返回FALSE
*)
METHOD Act_Extend : BOOL
VAR_INPUT
END_VAR
IF enable AND extCondition THEN// AND NOT busy
	Act_Extend:=extend:=TRUE;
ELSE
	Act_Extend:=FALSE;
END_IF
END_METHOD

(*
触发复位报警动作，成功触发返回TRUE，触发失败返回FALSE
*)
METHOD Act_Reset : BOOL
VAR_INPUT
END_VAR
Act_Reset:=reset:=TRUE;
END_METHOD

(*
触发缩回动作，成功触发返回TRUE，触发失败返回FALSE
*)
METHOD Act_Retract : BOOL
VAR_INPUT
END_VAR
IF enable AND retCondition THEN// AND NOT busy
	Act_Retract:=retract:=TRUE;
ELSE
	Act_Retract:=FALSE;
END_IF
END_METHOD

(*
触发停止输出动作，成功触发返回TRUE，触发失败返回FALSE
*)
METHOD Act_Stop : BOOL
VAR_INPUT
END_VAR
Act_Stop:=stop:=TRUE;
END_METHOD

ACTION Error_ACT:
CASE errorStep OF
	0:
		error:=FALSE;
		errID:=0;
		errTXT:='';
 (*
	1:
		error:=TRUE;
		errID:=errorID+errorStep;
		errTXT:=CONCAT(STR1:=nameTXT,STR2:=' Extend Error!');
		errWTXT:=WCONCAT(STR1:=TO_WSTRING(nameTXT),STR2:=" 伸出(打开)错误");
	2:
		error:=TRUE;
		errID:=errorID+errorStep;
		errTXT:=CONCAT(STR1:=nameTXT,STR2:=' Retract Error!');
		errWTXT:=WCONCAT(STR1:=TO_WSTRING(nameTXT),STR2:=" 缩回(关闭)错误");
		*)
	1..4:
		error:=TRUE;
		errID:=getErrID(errorStep);
		errTXT:=getErrTXT(errorStep);
		errWTXT:=getErrWTXT(errorStep);
END_CASE
END_ACTION

ACTION Extend_ACT:
// Chiller伸出--extend 触发
IF extend AND NOT extCondition THEN
	note_Ext:=TRUE;
	note_Ret:=FALSE;
	note_Set:=FALSE;
	NoteHMI.showFlag:=TRUE;
	NoteHMI.showText:='';
	NoteHMI.showText:=CONCAT(NoteHMI.showText,nameTXT);
	NoteHMI.showText:=CONCAT(NoteHMI.showText,' Open Condition Not Satisfied!');
	HMIItf.singleControl:=FALSE;
END_IF
IF extend AND enable AND extCondition THEN// AND NOT busy
	busy:=TRUE;
	retract:=FALSE;
	setPoint:=FALSE;
	setPoint:=FALSE;
	extdone:=FALSE;
	retdone:=FALSE;
	setdone:=FALSE;
	extStep:=10;
	retStep:=0;
	setStep:=0;
	note_Ext:=FALSE;
	note_Ret:=FALSE;
	note_Set:=FALSE;
	readAndWriteLock:=TRUE;
	//errorStep:=0;
END_IF
extend:=FALSE;
CASE extStep OF
0:
	//ready
	extErrorDelayTon(IN:=FALSE);
10:
	firstPower:=FALSE;
	extErrorDelayTon(IN:=FALSE);
	extDoneDelayTon(IN:=FALSE);
	extStep:=20;
	PLC_Chiller.readStartFlag:=FALSE;
	PLC_Chiller.WriteStart();
	extRelay:=TRUE;
	retRelay:=FALSE;
20:
	extErrorDelayTon(IN:=(NOT PLC_Chiller.readStartFlag),PT:=errorDelayTime);
	IF extErrorDelayTon.Q THEN
		//done:=FALSE;
		extdone:=FALSE;
		retdone:=FALSE;
		setdone:=FALSE;
		errorStep:=1;
		busy:=FALSE;
		readAndWriteLock:=FALSE;
		extStep:=40;
		extErrorDelayTon(IN:=FALSE);
		RETURN;
	END_IF
//	IF PLC_Chiller.readStartFlag THEN
//		extDoneDelayTon(IN:=PLC_Chiller.readStartFlag,PT:=doneDelayTimeShortExtend);
//	ELSE
//		extDoneDelayTon(IN:=NOT enableExtAprSw,PT:=doneDelayTimeLongExtend);
//	END_IF
	
	IF PLC_Chiller.readStartFlag THEN
		PLC_Chiller.readStartFlag:=FALSE;
		busy:=FALSE;
		//done:=TRUE;
		extdone:=TRUE;
		readAndWriteLock:=FALSE;
		retdone:=FALSE;
		errorStep:=0;
		IF NOT power THEN
			extRelay:=FALSE;
			retRelay:=FALSE;
		END_IF
		extStep:=30;
		extErrorDelayTon(IN:=FALSE);
	END_IF
END_CASE
END_ACTION

METHOD Get_Done_Ext : BOOL
VAR_INPUT
END_VAR
Get_Done_Ext:=extdone;
END_METHOD

METHOD Get_Done_Ret : BOOL
VAR_INPUT
END_VAR
Get_Done_Ret:=retdone;
END_METHOD

METHOD getErrID : UDINT
VAR_INPUT
	errID					:UDINT;//取值范围1~2
END_VAR
VAR
	nErrID					:UDINT;
END_VAR
nErrID:=errorID+errID;

getErrID:=nErrID;
END_METHOD

METHOD getErrTXT : STRING(255)
VAR_INPUT
	errID					:UDINT;//取值范围1~2
END_VAR
VAR
	sErrTXT					:STRING(255);
END_VAR

CASE errID OF
	1:
		sErrTXT:=CONCAT(STR1:=nameTXT,STR2:=' Extend Error!');
	2:
		sErrTXT:=CONCAT(STR1:=nameTXT,STR2:=' Retract Error!');
	3:
		sErrTXT:=CONCAT(STR1:=nameTXT,STR2:=' ParSet Error!');
	4:
		sErrTXT:=CONCAT(STR1:=nameTXT,STR2:=' State Error!');
ELSE
	sErrTXT:=CONCAT(STR1:=nameTXT,STR2:='');
END_CASE
getErrTXT:=sErrTXT;
END_METHOD

METHOD getErrWTXT : WSTRING(255)
VAR_INPUT
	errID					:UDINT;//取值范围1~16
END_VAR
VAR
	sErrTXT					:WSTRING(255);
END_VAR

CASE errID OF
	1:
		sErrTXT:=WCONCAT(STR1:=TO_WSTRING(nameTXT),STR2:=" 伸出(打开)错误");
	2:
		sErrTXT:=WCONCAT(STR1:=TO_WSTRING(nameTXT),STR2:=" 缩回(关闭)错误");
	3:
		sErrTXT:=WCONCAT(STR1:=TO_WSTRING(nameTXT),STR2:=" 参数设置错误");
ELSE
	sErrTXT:=WCONCAT(STR1:=TO_WSTRING(nameTXT),STR2:="");
END_CASE
getErrWTXT:=sErrTXT;
END_METHOD

ACTION Init_ACT:
done:=(extdone OR retdone);
InitHMI_ACT();
manualCtrl_ACT();
IF RTD1>alarmTemperatureH OR RTD1<alarmTemperatureL OR 
   RTD2>alarmTemperatureH OR RTD2<alarmTemperatureL THEN
   errorID:=4;
END_IF
noteTON_P(IN:=note_Ext,PT:=T#0.1S);
noteRTrig_P(CLK:=noteTON_P.Q);
IF noteRTrig_P.Q THEN
//	gLog_Note.append_EX(noteWTXT_Ext);
END_IF
noteTON_N(IN:=note_Ret,PT:=T#0.1S);
noteRTrig_N(CLK:=noteTON_N.Q);
IF noteRTrig_N.Q THEN
//	gLog_Note.append_EX(noteWTXT_Ret);
END_IF
extRealayRtrig(CLK:=extRelay);
IF extRealayRtrig.Q THEN
	HMIItf.singleControl:=TRUE;
END_IF
retRealayRtrig(CLK:=NOT extRelay);
IF retRealayRtrig.Q THEN
	HMIItf.singleControl:=FALSE;
END_IF
END_ACTION

ACTION InitHMI_ACT:
HMIItf.extAprSw:=extAprSw;
HMIItf.retAprSw:=retAprSw;
HMIItf.enableExt:=enableExtAprSw;
HMIItf.enableRet:=enableRetAprSw;
HMIItf.HMIEnable:=hmiEN;
HMIItf.enable:=enable;
HMIItf.done:=done;
HMIItf.busy:=busy;
HMIItf.error:=error;
HMIItf.errID:=UDINT_TO_DINT(errID);
HMIItf.errTXT:=errTXT;
HMIItf.extRelay:=extRelay;
HMIItf.retRelay:=retRelay;
HMIItf.power:=power;
HMIItf.nameTXT:=nameTXT;
HMIItf.extenderror:=error AND errorID=1;
HMIItf.retracterror:=error AND errorID=2;
HMIItf.extcondition:=extCondition;
HMIItf.retcondition:=retCondition;
HMIItf.sensorShow:=sensorShow;
END_ACTION

ACTION ManualCtrl_ACT:
//HMI手动控制
//IF ctrlMode=eManualCtrMode THEN
IF hmiEN THEN
	IF extAprSw AND extRelay THEN
		sensorShow:='UP';
	ELSIF retAprSw AND retRelay THEN
		sensorShow:='DOWN';
	ELSE
		sensorShow:='<->';
	END_IF
	extendTrigRAlc(CLK:=HMIItf.extendAndretract);
	IF extendTrigRAlc.Q THEN// AND NOT busy
		IF extRelay THEN//如果伸出继电器或伸出传感器亮，则认为已经伸出过
			retract:=TRUE;
		END_IF
		IF retRelay THEN
			extend:=TRUE;
		END_IF
		IF NOT extRelay AND NOT retRelay THEN
			IF extAprSw THEN
				retract:=TRUE;
			END_IF
			IF retAprSw THEN
				extend:=TRUE;
			END_IF
		END_IF
	END_IF
	singleControlR(CLK:=HMIItf.singleControltemp);
	singleControlF(CLK:=HMIItf.singleControl);
	
	extendTrigR1(CLK:=HMIItf.extend );
	IF extendTrigR1.Q OR (singleControlR.Q AND NOT HMIItf.singleControl) THEN// AND NOT busy
		WarmHMI.showText:='';
		WarmHMI.showFlag:=TRUE;
		WarmHMI.showText:=CONCAT(WarmHMI.showText,'Are you sure you want to Extend the ');
		WarmHMI.showText:=CONCAT(WarmHMI.showText,nameTXT);
		WarmHMI.showText:=CONCAT(WarmHMI.showText,' ?');
	END_IF
	IF WarmHMI.bOK AND NOT WarmHMI.showFlag AND FIND(WarmHMI.showText,nameTXT)>0 AND FIND(WarmHMI.showText,'Extend')>0 THEN
		IF HMIItf.singleControl THEN
			;
		ELSE
			extend:=TRUE;
			operatorLog.append(CONCAT(nameTXT,' Extend'));
		END_IF
		HMIItf.singleControl:= NOT HMIItf.singleControl;
		WarmHMI.bOK:=FALSE;
		WarmHMI.showText:='';
	END_IF
	IF WarmHMI.bNO AND NOT WarmHMI.showFlag AND FIND(WarmHMI.showText,nameTXT)>0 AND FIND(WarmHMI.showText,'Extend')>0 THEN
		WarmHMI.bNO:=FALSE;
		HMIItf.extend:=FALSE;
		WarmHMI.showText:='';
	END_IF
	
	retractTrigR1(CLK:=HMIItf.retract);
	IF retractTrigR1.Q OR (singleControlR.Q AND HMIItf.singleControl) THEN// AND NOT busy
		WarmHMI.showText:='';
		WarmHMI.showFlag:=TRUE;
		WarmHMI.showText:=CONCAT(WarmHMI.showText,'Are you sure you want to Retract the ');
		WarmHMI.showText:=CONCAT(WarmHMI.showText,nameTXT);
		WarmHMI.showText:=CONCAT(WarmHMI.showText,' ?');
	END_IF
		IF WarmHMI.bOK AND NOT WarmHMI.showFlag AND FIND(WarmHMI.showText,nameTXT)>0 AND FIND(WarmHMI.showText,'Retract')>0 THEN
		IF HMIItf.singleControl THEN
			retract:=TRUE;
			operatorLog.append(CONCAT(nameTXT,' Retract'));
		ELSE
			;
		END_IF
		HMIItf.singleControl:= NOT HMIItf.singleControl;
		WarmHMI.bOK:=FALSE;
		WarmHMI.showText:='';
	END_IF
	IF WarmHMI.bNO AND NOT WarmHMI.showFlag AND FIND(WarmHMI.showText,nameTXT)>0 AND FIND(WarmHMI.showText,'Retract')>0 THEN
		WarmHMI.bNO:=FALSE;
		HMIItf.singleControl:=FALSE;
		HMIItf.retract:=FALSE;
		WarmHMI.showText:='';
	END_IF
	
	setR(CLK:=HMIItf.set);
	IF setR.Q THEN
		WarmHMI.showText:='';
		WarmHMI.showFlag:=TRUE;
		WarmHMI.showText:=CONCAT(WarmHMI.showText,'Are you sure you want ');
		WarmHMI.showText:=CONCAT(WarmHMI.showText,nameTXT);
		WarmHMI.showText:=CONCAT(WarmHMI.showText,' to Set it?');
		HMIItf.set:=FALSE;
	END_IF
		IF WarmHMI.bOK AND NOT WarmHMI.showFlag AND FIND(WarmHMI.showText,nameTXT)>0 AND FIND(WarmHMI.showText,'Set')>0 THEN
		setPoint:=TRUE;
		operatorLog.append(CONCAT(nameTXT,' Set'));
		WarmHMI.bOK:=FALSE;
		WarmHMI.showText:='';
	END_IF
	IF WarmHMI.bNO AND NOT WarmHMI.showFlag AND FIND(WarmHMI.showText,nameTXT)>0 AND FIND(WarmHMI.showText,'Set')>0 THEN
		WarmHMI.bNO:=FALSE;
		HMIItf.singleControl:=FALSE;
		WarmHMI.showText:='';
	END_IF
	
	resetTrigR1(CLK:=HMIItf.reset);
	IF resetTrigR1.Q THEN// AND NOT busy
		reset:=TRUE;
	END_IF
	
	stopTrigR1(CLK:=HMIItf.stop);
	IF stopTrigR1.Q THEN// AND NOT busy
		stop:=TRUE;
	END_IF
	
	powerTrigR1(CLK:=HMIItf.power);
	IF powerTrigR1.Q THEN// AND NOT busy
		IF power THEN
			power:=FALSE;
		ELSE
			power:=TRUE;
		END_IF
	END_IF
END_IF
END_ACTION

ACTION Read_ACT:
//气缸收回--read 触发
IF NOT readAndWriteLock AND NOT busy AND NOT readbusy AND readStep=0 AND readCondition THEN// AND NOT busy
	retdone:=FALSE;
	retStep:=0;
	extStep:=0;
	setStep:=0;
	readStep:=10;
	setStep:=0;
	readbusy:=TRUE;
	readerror:=FALSE;
END_IF
CASE readStep OF
0:
	//ready
	readTon1(IN:=FALSE);
	readTon2(IN:=FALSE);
10:// State
	IF readAndWriteLock THEN
		readStep:=5000;
	ELSE
		PLC_Chiller.readStateFlag:=FALSE;
		PLC_Chiller.ReadState();
		readStep:=readStep+10;
	END_IF
20:
	IF readAndWriteLock THEN
		readStep:=5000;
	ELSE
		IF PLC_Chiller.readStateFlag THEN
			PLC_Chiller.readStateFlag:=FALSE;
			// 数据处理
			readTon1(IN:=FALSE);
			readStep:=100;
			RETURN;
		END_IF
		readTon1(IN:=TRUE,PT:=T#500MS);// 超时
		IF readTon1.Q THEN
			readStep:=6000;
			readTon1(IN:=FALSE);
			readTon2(IN:=FALSE);
			RETURN;
		END_IF
		;
	END_IF
100:// Internal RTD1
	IF readAndWriteLock THEN
		readStep:=5000;
	ELSE
		PLC_Chiller.readRTD1Flag:=FALSE;
		PLC_Chiller.ReadRTD1();
		readStep:=readStep+10;
	END_IF	
110:
	IF readAndWriteLock THEN
		readStep:=5000;
	ELSE
		IF PLC_Chiller.readRTD1Flag THEN
			PLC_Chiller.readRTD1Flag:=FALSE;
			// 数据处理
			readTon1(IN:=FALSE);
			readStep:=200;
			RETURN;
		END_IF
		readTon1(IN:=TRUE,PT:=T#500MS);// 超时
		IF readTon1.Q THEN
			readStep:=6000;
			readTon1(IN:=FALSE);
			readTon2(IN:=FALSE);
			RETURN;
		END_IF
		;
	END_IF
	
200:// External RTD2
	IF readAndWriteLock THEN
		readStep:=5000;
	ELSE
		PLC_Chiller.readRTD2Flag:=FALSE;
		PLC_Chiller.ReadRTD2();
		readStep:=readStep+10;
	END_IF
210:
	IF readAndWriteLock THEN
		readStep:=5000;
	ELSE
		IF PLC_Chiller.readRTD2Flag THEN
			PLC_Chiller.readRTD2Flag:=FALSE;
			// 数据处理
			readTon1(IN:=FALSE);
			readStep:=5000;
			RETURN;
		END_IF
		readTon1(IN:=TRUE,PT:=T#500MS);// 超时
		IF readTon1.Q THEN
			readStep:=6000;
			readTon1(IN:=FALSE);
			readTon2(IN:=FALSE);
			RETURN;
		END_IF
		;
	END_IF
5000:
	readbusy:=FALSE;
	readdone:=TRUE;
	readStep:=0;
	readerror:=FALSE;
6000:
	readbusy:=FALSE;
	readdone:=TRUE;
	readStep:=0;
	readerror:=TRUE;
END_CASE
END_ACTION

ACTION Reset_ACT:
IF reset THEN
	IF NOT power THEN
		extRelay:=FALSE;
		retRelay:=FALSE;
	END_IF
	busy:=FALSE;
	//done:=FALSE;
	//extdone:=FALSE;
	//retdone:=FALSE;
	errorStep:=0;
	note_Ext:=FALSE;
	note_Ret:=FALSE;
	note_Set:=FALSE;
	reset:=FALSE;
END_IF

IF stop THEN
	stop:=FALSE;
	extRelay:=FALSE;
	retRelay:=FALSE;
	note_Ext:=FALSE;
	note_Ret:=FALSE;
	//无自锁检测说法，直接停
//	extStep:=0;
//	retStep:=0;
END_IF
END_ACTION

ACTION Retract_ACT:
//Chiller收回--retract 触发
IF retract AND NOT retCondition THEN
	note_Ret:=TRUE;
	note_Ext:=FALSE;
	note_Set:=FALSE;
	NoteHMI.showFlag:=TRUE;
	NoteHMI.showText:='';
	NoteHMI.showText:=CONCAT(NoteHMI.showText,nameTXT);
	NoteHMI.showText:=CONCAT(NoteHMI.showText,' Close Condition Not Satisfied!');
END_IF
IF retract AND enable AND retCondition THEN// AND NOT busy
	busy:=TRUE;
	extend:=FALSE;
	setPoint:=FALSE;
	setPoint:=FALSE;
	extdone:=FALSE;
	retdone:=FALSE;
	setdone:=FALSE;
	retStep:=10;
	extStep:=0;
	setStep:=0;
	note_Ext:=FALSE;
	note_Ret:=FALSE;
	note_Set:=FALSE;
	readAndWriteLock:=TRUE;
END_IF
retract:=FALSE;
CASE retStep OF
0:
	//ready
	retErrorDelayTon(IN:=FALSE);
10:
	firstPower:=FALSE;
	retErrorDelayTon(IN:=FALSE);
	retDoneDelayTon(IN:=FALSE);
	retStep:=20;
	PLC_Chiller.readStopFlag:=FALSE;
	PLC_Chiller.WriteStop();
	extRelay:=FALSE;
	retRelay:=TRUE;
20:
	retErrorDelayTon(IN:=(NOT PLC_Chiller.readStopFlag),PT:=errorDelayTime);
	IF retErrorDelayTon.Q THEN
		//done:=FALSE;
		extdone:=FALSE;
		retdone:=FALSE;
		setdone:=FALSE;
		errorStep:=2;
		busy:=FALSE;
		readAndWriteLock:=FALSE;
		retStep:=40;
		retErrorDelayTon(IN:=FALSE);
		RETURN;
	END_IF
//	IF enableRetAprSw THEN
//		retDoneDelayTon(IN:=retAprSw,PT:=doneDelayTimeShortRetract);
//	ELSE
//		retDoneDelayTon(IN:=NOT enableRetAprSw,PT:=doneDelayTimeLongRetract);
//	END_IF
	
	IF PLC_Chiller.readStopFlag THEN
		busy:=FALSE;
		//done:=TRUE;
		extdone:=FALSE;
		retdone:=TRUE;
		readAndWriteLock:=FALSE;
		errorStep:=0;
		IF NOT power  THEN
			extRelay:=FALSE;
			retRelay:=FALSE;
		END_IF
		retStep:=30;
		retErrorDelayTon(IN:=FALSE);
	END_IF
END_CASE
END_ACTION

ACTION SafeMonitor_ACT:
//notBusyMonitorDelayTon(IN:=NOT busy,PT:=notBusyMonitorDelayTime);
//IF real_TimeMonitor THEN
//	IF notBusyMonitorDelayTon.Q THEN
//		//伸出实时检测
//		IF (enableExtAprSw AND NOT extAprSw) AND extRelay THEN
//			errorStep:=1;
//		END_IF
	
//		//缩回实时检测	
//		IF (enableRetAprSw AND NOT retAprSw) AND retRelay  THEN
//			errorStep:=2;
//		END_IF
//	END_IF
//END_IF
END_ACTION

ACTION Set_ACT:
//Chiller收回--retract 触发
IF setPoint AND NOT setCondition THEN
	note_Set:=TRUE;
	note_Ext:=FALSE;
	note_Ret:=FALSE;
	NoteHMI.showFlag:=TRUE;
	NoteHMI.showText:='';
	NoteHMI.showText:=CONCAT(NoteHMI.showText,nameTXT);
	NoteHMI.showText:=CONCAT(NoteHMI.showText,' Set Par Condition Not Satisfied!');
END_IF
IF setPoint AND enable AND setCondition THEN// AND NOT busy
	busy:=TRUE;
	extend:=FALSE;
	retract:=FALSE;
	setPoint:=FALSE;
	extdone:=FALSE;
	retdone:=FALSE;
	setdone:=FALSE;
	retStep:=0;
	extStep:=0;
	setStep:=0;
	setStep:=10;
	note_Ext:=FALSE;
	note_Ret:=FALSE;
	note_Set:=FALSE;
	readAndWriteLock:=TRUE;
END_IF
setPoint:=FALSE;
CASE setStep OF
0:
	//ready
	setErrorDelayTon(IN:=FALSE);
10:
	firstPower:=FALSE;
	setErrorDelayTon(IN:=FALSE);
	setDoneDelayTon(IN:=FALSE);
	setStep:=20;

	PLC_Chiller.readSetAckFlag:=FALSE;
	PLC_Chiller.WriteTemperature(setpointVal);
20:
	setErrorDelayTon(IN:=(NOT PLC_Chiller.readSetAckFlag),PT:=errorDelayTime);
	IF setErrorDelayTon.Q THEN
		//done:=FALSE;
		extdone:=FALSE;
		retdone:=FALSE;
		setdone:=FALSE;
		errorStep:=3;
		busy:=FALSE;
		readAndWriteLock:=FALSE;
		setStep:=40;
		setErrorDelayTon(IN:=FALSE);
		RETURN;
	END_IF
	IF PLC_Chiller.readSetAckFlag THEN
		PLC_Chiller.readSetAckFlag:=FALSE;
		setStep:=30;
		busy:=FALSE;
		//done:=TRUE;
		extdone:=FALSE;
		retdone:=FALSE;
		setdone:=TRUE;
		readAndWriteLock:=FALSE;
		errorStep:=0;
		setErrorDelayTon(IN:=FALSE);
		IF NOT power  THEN
			extRelay:=FALSE;
			retRelay:=FALSE;
		END_IF
	END_IF
	;
END_CASE
END_ACTION

ACTION VersionLog:
(*
版本: V1.0.0.0
说明:
	1. 首个版本
	2. 含普通气缸\真空吸类型的控制
	3. 可配置是否有到位信号, 以及到位稳定时间
(--------------------------------------------------)
新版本: V1.0.1.0
更新时间: 2019/11/20 19:00
更新说明:
	1. 优化编写方式
	2. 修改错误编码起始位，现改为从1开始
(--------------------------------------------------)
新版本: V1.0.1.1
更新时间: 2020/03/23 23:00
更新说明:
	1. 优化报错方式
	2. 增加伸出、缩回、复位和停止触发函数
(--------------------------------------------------)
新版本: V1.0.1.2
更新时间: 2020/04/22 09:50
更新说明:
	1. 增加中文报警输出
(--------------------------------------------------)
新版本: V1.0.1.3
更新时间: 2020/09/16
更新说明:
	1. 开放错误ID、错误文本信息获取接口
(--------------------------------------------------)
新版本: V1.0.1.4
更新时间: 2020/10/06
更新说明:
	1. 移除控制模式变量，增加HMI启用条件
	2. 增加外部获取伸出缩回完成信号接口函数
(--------------------------------------------------)
新版本: V1.0.1.5
更新时间: 2020/10/14
更新说明:
	1. 优化代码
(--------------------------------------------------)
*)
END_ACTION

END_FUNCTION_BLOCK

// ---- POUs/Communication/PLC_Chiller.TcPOU
PROGRAM PLC_Chiller
VAR_INPUT
	nSocketType:UINT:=1;// socket 类型; 0 表示 server; 1 表示 client;
	sTerminalName:STRING;// 通讯对方名称 自定义
	sHost:STRING(20):='127.0.0.1';// 通讯IP地址; server时表示本地host; client时表示远程host
	nPort:UDINT:=8900;// 通讯端口号;
	bEnable:BOOL:=TRUE;// 通讯启用\禁用连接
	sSendSuffix:STRING:='';//此处可统一添加发送后缀字符 $R$N
	nQueueInterval:UDINT:=50;// 发送队列时间间隔 单位ms
	logHandleArray:ARRAY [1..5] OF POINTER TO printLogModule_EX;// log 操作 handle 数组
	logHandleArrayLength:UINT:=0;// log 操作 handle 数组长度, 不超过5
	enHeartBeat:BOOL;// 启用心跳包命令
	cmdHeartBeat:DINT;// 心跳包命令
	readStateFlag:BOOL;
	readRTD1Flag:BOOL;
	readRTD2Flag:BOOL;
	readStartFlag:BOOL;
	readStopFlag:BOOL;
	readSetAckFlag:BOOL;
END_VAR
VAR_OUTPUT
	bSendCondition	:BOOL;//可发送条件
	bSocketConnected:BOOL;//连接状态
	
END_VAR
VAR CONSTANT
	cNumBegin		:DINT:=1;
	cNumEnd			:DINT:=100;
END_VAR
VAR
	sendDataArray	:ARRAY [cNumBegin..cNumEnd] OF struct_byte;
	length			:DINT:=0;
	endPoint		:DINT:=cNumBegin;
	sendPoint		:DINT:=cNumBegin;
	passMax			:BOOL;
	popupSendData	:struct_byte;
	//popup
	popupStep		:UINT:=0;
	popupTON1		:TON;
	popupTON2		:TON;
	iPopup			:DINT:=0;
	_PopupLength	:DINT:=0;
	sendDataTemp	:struct_byte;
	sendLenght		:UDINT;
END_VAR
VAR
	tcpipClient					:tcpipClientModule_EX;
	tcpipServer					:tcpipServerModule_EX;////定义服务器对象
	
	tcpipSendDataBuff_Server	:struct_byte;//发送数据 Buff server
	tcpipSendDataBuff_Client	:struct_byte;//发送数据 Buff client
	
	tcpipSendDataClear			:struct_byte;//发送数据 清空
	tcpipSendData				:struct_byte;//发送数据
	
	tcpipRecDataBuff_Server		:struct_byte;//已接收数据 Buff server
	tcpipRecDataBuff_Client		:struct_byte;//已接收数据 Buff client
	
	tcpipRecDataClear			:struct_byte;//已接收数据 清空
	tcpipRecData				:struct_byte;//已接收数据
	
	tcpConnectR_Trig			:R_Trig;//初始连接上升沿
	tcpConnectF_Trig			:F_Trig;//初始连接下降沿
	registerStep				:UDINT;//ALC注册控制步
	registerTON					:TON;//ALC注册延时
	
	logHandleArray_index		:UINT:=1;
END_VAR
VAR
	(*
	bTrig_Version:BOOL;
	rTrig_Version:R_TRIG;
	*)
END_VAR


CASE nSocketType OF
0://TCPIP server
	tcpipServer(
		sSrvNetId:= , 
		sLocalHost:=sHost , 
		nLocalPort:=nPort , 
		bStartConnect:=bEnable , 
		tcpipSDataLen:=sendLenght , 
		tcpipSData:=ADR(tcpipSendDataBuff_Server) , 
		bSend:= , 
		tcpipRecDataLen:=SIZEOF(tcpipRecDataBuff_Server), 
		tcpipRecData:=ADR(tcpipRecDataBuff_Server) , 
		bAccepted=> , 
		bSendBusy=> , 
		bRecData=> );
	bSendCondition:=tcpipServer.bAccepted AND NOT tcpipServer.bSendBusy;
	//TCPIP连接
	bSocketConnected:=tcpipServer.bAccepted;
	IF NOT tcpipServer.bAccepted THEN
		length:=0;
		endPoint:=cNumBegin;
		sendPoint:=cNumBegin;
		passMax:=FALSE;
	END_IF
	tcpConnectR_Trig(CLK:=tcpipServer.bAccepted);
	tcpConnectF_Trig(CLK:=tcpipServer.bAccepted);

1://TCPIP client
	tcpipClient(
		sSrvNetId:= , 
		sRemoteHost:=sHost , 
		nRemotePort:=nPort , 
		bStartConnect:=bEnable , 
		tcpipSDataLen:=sendLenght, 
		tcpipSData:=ADR(tcpipSendDataBuff_Client) , 
		bSend:= , 
		tcpipRecDataLen:=SIZEOF(tcpipRecDataBuff_Client) , 
		tcpipRecData:=ADR(tcpipRecDataBuff_Client) , 
		bConnected=> , 
		bSendBusy=> , 
		bRecData=> );
	bSendCondition:=tcpipClient.bConnected AND NOT tcpipClient.bSendBusy;
	//TCPIP连接
	bSocketConnected:=tcpipClient.bConnected;
	IF NOT tcpipClient.bConnected THEN
		length:=0;
		endPoint:=cNumBegin;
		sendPoint:=cNumBegin;
		passMax:=FALSE;
	END_IF
	tcpConnectR_Trig(CLK:=tcpipClient.bConnected);
	tcpConnectF_Trig(CLK:=tcpipClient.bConnected);
END_CASE

IF tcpConnectR_Trig.Q THEN
	FOR logHandleArray_index:=1 TO logHandleArrayLength DO
		logHandleArray[logHandleArray_index]^.append(CONCAT(sTerminalName, ' has been connected'));
	END_FOR
	registerStep:=10;
END_IF
IF tcpConnectF_Trig.Q THEN
	FOR logHandleArray_index:=1 TO logHandleArrayLength DO
		logHandleArray[logHandleArray_index]^.append(CONCAT(sTerminalName, ' has been disconnected'));
	END_FOR
	registerStep:=0;
END_IF
//数据接收处理
CASE nSocketType OF
0://TCPIP server
	IF tcpipServer.bRecData THEN
		tcpipRecData:=tcpipRecDataBuff_Server;//buff转存
		tcpipRecDataBuff_Server:=tcpipRecDataClear;//转存之后清空buff
		dataProcessing();
	END_IF
1://TCPIP client
	IF tcpipClient.bRecData THEN
		tcpipRecData:=tcpipRecDataBuff_Client;//buff转存
		tcpipRecDataBuff_Client:=tcpipRecDataClear;//转存之后清空buff
		dataProcessing();
	END_IF
END_CASE


popup();

CASE registerStep OF
0:
	//Ready
10:
	registerStep:=0;
// 心跳包
20:
	IF NOT enHeartBeat THEN
		registerStep:=0;
	ELSE
		registerStep:=registerStep+10;
	END_IF
30:
	registerTON(IN:=FALSE);
	appendSend(1,1,1,1,1,1,1,1,1,1,1,1,1,1,1,1,1,1,1,1,20);
	registerStep:=registerStep+10;
40:
	registerTON(IN:=NOT registerTON.Q,PT:=T#3S);
	IF registerTON.Q THEN
		registerTON(IN:=FALSE);
		registerStep:=30;
	END_IF
END_CASE

Manual();

METHOD appendSend : BOOL
VAR_INPUT
	b1		:BYTE:=0;
	b2		:BYTE:=0;
	b3		:Byte:=0;
	b4		:Byte:=0;
	b5		:Byte:=0;
	b6		:Byte:=0;
	b7		:Byte:=0;
	b8		:Byte:=0;
	b9		:BYTE:=0;
	b10		:BYTE:=0;
	b11		:BYTE:=0;
	b12		:BYTE:=0;
	b13		:BYTE:=0;
	b14		:BYTE:=0;
	b15		:BYTE:=0;
	b16		:BYTE:=0;
	b17		:BYTE:=0;
	b18		:BYTE:=0;
	b19		:BYTE:=0;
	b20		:BYTE:=0;
	lenght	:UDINT;
END_VAR
sendLenght:=lenght;
sendDataArray[endPoint].b1:=b1;
sendDataArray[endPoint].b2:=b2;
sendDataArray[endPoint].b3:=b3;
sendDataArray[endPoint].b4:=b4;
sendDataArray[endPoint].b5:=b5;
sendDataArray[endPoint].b6:=b6;
sendDataArray[endPoint].b7:=b7;
sendDataArray[endPoint].b8:=b8;
sendDataArray[endPoint].b9:=b9;
sendDataArray[endPoint].b10:=b10;
sendDataArray[endPoint].b11:=b11;
sendDataArray[endPoint].b12:=b12;
sendDataArray[endPoint].b13:=b13;
sendDataArray[endPoint].b14:=b14;
sendDataArray[endPoint].b15:=b15;
sendDataArray[endPoint].b16:=b16;
sendDataArray[endPoint].b17:=b17;
sendDataArray[endPoint].b18:=b18;
sendDataArray[endPoint].b19:=b19;
sendDataArray[endPoint].b20:=b20;

endPoint:=endPoint+1;
IF endPoint>(cNumEnd-1) THEN
	endPoint:=1;
	passMax:=TRUE;
END_IF
END_METHOD

METHOD dataProcessing : BOOL
VAR_INPUT
END_VAR
VAR
	i_CGResult:INT;
	i_HResult:INT;
	str1:STRING;
END_VAR
FOR logHandleArray_index:=1 TO logHandleArrayLength DO
	CASE nSocketType OF
	0://TCPIP server
		str1:=CONCAT(str1,BYTE_TO_HEXSTR(tcpipRecData.b1,2,FALSE));
		str1:=CONCAT(str1,' ');
		str1:=CONCAT(str1,BYTE_TO_HEXSTR(tcpipRecData.b2,2,FALSE));
		str1:=CONCAT(str1,' ');
		str1:=CONCAT(str1,BYTE_TO_HEXSTR(tcpipRecData.b3,2,FALSE));
		str1:=CONCAT(str1,' ');
		str1:=CONCAT(str1,BYTE_TO_HEXSTR(tcpipRecData.b4,2,FALSE));
		str1:=CONCAT(str1,' ');
		str1:=CONCAT(str1,BYTE_TO_HEXSTR(tcpipRecData.b5,2,FALSE));
		str1:=CONCAT(str1,' ');
		str1:=CONCAT(str1,BYTE_TO_HEXSTR(tcpipRecData.b6,2,FALSE));
		str1:=CONCAT(str1,' ');
		str1:=CONCAT(str1,BYTE_TO_HEXSTR(tcpipRecData.b7,2,FALSE));
		str1:=CONCAT(str1,' ');
		str1:=CONCAT(str1,BYTE_TO_HEXSTR(tcpipRecData.b8,2,FALSE));
		str1:=CONCAT(str1,' ');
		str1:=CONCAT(str1,BYTE_TO_HEXSTR(tcpipRecData.b9,2,FALSE));
		str1:=CONCAT(str1,' ');
		str1:=CONCAT(str1,BYTE_TO_HEXSTR(tcpipRecData.b10,2,FALSE));
		str1:=CONCAT(str1,' ');
		str1:=CONCAT(str1,BYTE_TO_HEXSTR(tcpipRecData.b11,2,FALSE));
		str1:=CONCAT(str1,' ');
		str1:=CONCAT(str1,BYTE_TO_HEXSTR(tcpipRecData.b12,2,FALSE));
		str1:=CONCAT(str1,' ');
		str1:=CONCAT(str1,BYTE_TO_HEXSTR(tcpipRecData.b13,2,FALSE));
		str1:=CONCAT(str1,' ');
		str1:=CONCAT(str1,BYTE_TO_HEXSTR(tcpipRecData.b14,2,FALSE));
		str1:=CONCAT(str1,' ');
		str1:=CONCAT(str1,BYTE_TO_HEXSTR(tcpipRecData.b15,2,FALSE));
		str1:=CONCAT(str1,' ');
		str1:=CONCAT(str1,BYTE_TO_HEXSTR(tcpipRecData.b16,2,FALSE));
		str1:=CONCAT(str1,' ');
		str1:=CONCAT(str1,BYTE_TO_HEXSTR(tcpipRecData.b17,2,FALSE));
		str1:=CONCAT(str1,' ');
		str1:=CONCAT(str1,BYTE_TO_HEXSTR(tcpipRecData.b18,2,FALSE));
		str1:=CONCAT(str1,' ');
		str1:=CONCAT(str1,BYTE_TO_HEXSTR(tcpipRecData.b19,2,FALSE));
		str1:=CONCAT(str1,' ');
		str1:=CONCAT(str1,BYTE_TO_HEXSTR(tcpipRecData.b20,2,FALSE));
		logHandleArray[logHandleArray_index]^.append(CONCAT(CONCAT(CONCAT('Recevie From ', sTerminalName), ' -- '),str1));
	1://TCPIP client
		str1:=CONCAT(str1,BYTE_TO_HEXSTR(tcpipRecData.b1,2,FALSE));
		str1:=CONCAT(str1,' ');
		str1:=CONCAT(str1,BYTE_TO_HEXSTR(tcpipRecData.b2,2,FALSE));
		str1:=CONCAT(str1,' ');
		str1:=CONCAT(str1,BYTE_TO_HEXSTR(tcpipRecData.b3,2,FALSE));
		str1:=CONCAT(str1,' ');
		str1:=CONCAT(str1,BYTE_TO_HEXSTR(tcpipRecData.b4,2,FALSE));
		str1:=CONCAT(str1,' ');
		str1:=CONCAT(str1,BYTE_TO_HEXSTR(tcpipRecData.b5,2,FALSE));
		str1:=CONCAT(str1,' ');
		str1:=CONCAT(str1,BYTE_TO_HEXSTR(tcpipRecData.b6,2,FALSE));
		str1:=CONCAT(str1,' ');
		str1:=CONCAT(str1,BYTE_TO_HEXSTR(tcpipRecData.b7,2,FALSE));
		str1:=CONCAT(str1,' ');
		str1:=CONCAT(str1,BYTE_TO_HEXSTR(tcpipRecData.b8,2,FALSE));
		str1:=CONCAT(str1,' ');
		str1:=CONCAT(str1,BYTE_TO_HEXSTR(tcpipRecData.b9,2,FALSE));
		str1:=CONCAT(str1,' ');
		str1:=CONCAT(str1,BYTE_TO_HEXSTR(tcpipRecData.b10,2,FALSE));
		str1:=CONCAT(str1,' ');
		str1:=CONCAT(str1,BYTE_TO_HEXSTR(tcpipRecData.b11,2,FALSE));
		str1:=CONCAT(str1,' ');
		str1:=CONCAT(str1,BYTE_TO_HEXSTR(tcpipRecData.b12,2,FALSE));
		str1:=CONCAT(str1,' ');
		str1:=CONCAT(str1,BYTE_TO_HEXSTR(tcpipRecData.b13,2,FALSE));
		str1:=CONCAT(str1,' ');
		str1:=CONCAT(str1,BYTE_TO_HEXSTR(tcpipRecData.b14,2,FALSE));
		str1:=CONCAT(str1,' ');
		str1:=CONCAT(str1,BYTE_TO_HEXSTR(tcpipRecData.b15,2,FALSE));
		str1:=CONCAT(str1,' ');
		str1:=CONCAT(str1,BYTE_TO_HEXSTR(tcpipRecData.b16,2,FALSE));
		str1:=CONCAT(str1,' ');
		str1:=CONCAT(str1,BYTE_TO_HEXSTR(tcpipRecData.b17,2,FALSE));
		str1:=CONCAT(str1,' ');
		str1:=CONCAT(str1,BYTE_TO_HEXSTR(tcpipRecData.b18,2,FALSE));
		str1:=CONCAT(str1,' ');
		str1:=CONCAT(str1,BYTE_TO_HEXSTR(tcpipRecData.b19,2,FALSE));
		str1:=CONCAT(str1,' ');
		str1:=CONCAT(str1,BYTE_TO_HEXSTR(tcpipRecData.b20,2,FALSE));
		logHandleArray[logHandleArray_index]^.append(CONCAT(CONCAT(CONCAT('Recevie From ', sTerminalName), ' -- '),str1));
	END_CASE
END_FOR

// 数据处理
IF tcpipRecData.b4=16#09 THEN
	readStateFlag:=TRUE;
	gICP.Chiller.pumon:=tcpipRecData.b9.2;// Pum on
	gICP.Chiller.uinton:=tcpipRecData.b9.3;// Unit on
	gICP.Chiller.unitstoping:=tcpipRecData.b9.4;// Unit stopping
	gICP.Chiller.fault:=tcpipRecData.b9.4;// Fault
END_IF
IF tcpipRecData.b4=16#81 THEN
	IF tcpipRecData.b6=16#01 THEN
		readStartFlag:=TRUE;
	END_IF
	IF tcpipRecData.b6=16#00 THEN
		readStopFlag:=TRUE;
	END_IF
END_IF
IF tcpipRecData.b4=16#F0 THEN
	readSetAckFlag:=TRUE;
END_IF
IF tcpipRecData.b4=16#20 THEN
	readRTD1Flag:=TRUE;
	CASE tcpipRecData.b6 OF
	16#00:
		gICP.Chiller.RTD1:=(BYTE_TO_INT(tcpipRecData.b7)*256+BYTE_TO_INT(tcpipRecData.b8))*1.0;
	16#01:
		gICP.Chiller.RTD1:=(BYTE_TO_INT(tcpipRecData.b7)*256+BYTE_TO_INT(tcpipRecData.b8))*0.1;
	16#20:	
		gICP.Chiller.RTD1:=(BYTE_TO_INT(tcpipRecData.b7)*256+BYTE_TO_INT(tcpipRecData.b8))*0.01;
	16#11:
		gICP.Chiller.RTD1:=(BYTE_TO_INT(tcpipRecData.b7)*256+BYTE_TO_INT(tcpipRecData.b8))*1.0;
	16#21:
		gICP.Chiller.RTD1:=(BYTE_TO_INT(tcpipRecData.b7)*256+BYTE_TO_INT(tcpipRecData.b8))*0.1;
	16#22:	
		gICP.Chiller.RTD1:=(BYTE_TO_INT(tcpipRecData.b7)*256+BYTE_TO_INT(tcpipRecData.b8))*0.01;
	16#1D:
		gICP.Chiller.RTD1:=(BYTE_TO_INT(tcpipRecData.b7)*256+BYTE_TO_INT(tcpipRecData.b8))*0.1;
	16#2D:	
		gICP.Chiller.RTD1:=(BYTE_TO_INT(tcpipRecData.b7)*256+BYTE_TO_INT(tcpipRecData.b8))*0.01;
	END_CASE
END_IF
IF tcpipRecData.b4=16#21 THEN
	readRTD2Flag:=TRUE;
	CASE tcpipRecData.b6 OF
	16#00:
		gICP.Chiller.RTD2:=(BYTE_TO_INT(tcpipRecData.b7)*256+BYTE_TO_INT(tcpipRecData.b8))*1.0;
	16#01:
		gICP.Chiller.RTD2:=(BYTE_TO_INT(tcpipRecData.b7)*256+BYTE_TO_INT(tcpipRecData.b8))*0.1;
	16#20:	
		gICP.Chiller.RTD2:=(BYTE_TO_INT(tcpipRecData.b7)*256+BYTE_TO_INT(tcpipRecData.b8))*0.01;
	16#11:
		gICP.Chiller.RTD2:=(BYTE_TO_INT(tcpipRecData.b7)*256+BYTE_TO_INT(tcpipRecData.b8))*1.0;
	16#21:
		gICP.Chiller.RTD2:=(BYTE_TO_INT(tcpipRecData.b7)*256+BYTE_TO_INT(tcpipRecData.b8))*0.1;
	16#22:	
		gICP.Chiller.RTD2:=(BYTE_TO_INT(tcpipRecData.b7)*256+BYTE_TO_INT(tcpipRecData.b8))*0.01;
	16#1D:
		gICP.Chiller.RTD2:=(BYTE_TO_INT(tcpipRecData.b7)*256+BYTE_TO_INT(tcpipRecData.b8))*0.1;
	16#2D:	
		gICP.Chiller.RTD2:=(BYTE_TO_INT(tcpipRecData.b7)*256+BYTE_TO_INT(tcpipRecData.b8))*0.01;
	END_CASE
END_IF
END_METHOD

ACTION Manual:
(*
rTrig_Version(CLK:=bTrig_Version);
IF rTrig_Version.Q THEN
	appendSend(0,0,E_CmdID_SW.SW_GetVer,0.0,0.0,0.0,0.0,0.0,0,'');
END_IF
*)
END_ACTION

METHOD PRIVATE popup : BOOL
VAR_INPUT
END_VAR
CASE popupStep OF
0:
	IF (sendPoint<endPoint OR passMax) AND bSendCondition THEN
		popupSendData:=sendDataArray[sendPoint];
		sendData(popupSendData);//此处是调用信息发送
		popupStep:=10;
		sendPoint:=sendPoint+1;
		IF sendPoint>(cNumEnd-1) THEN
			sendPoint:=1;
			passMax:=FALSE;
		END_IF
	END_IF
10:
	popupTON2(IN:=NOT popupTON2.Q, PT:=T#2S);
	IF NOT bSendCondition OR popupTON2.Q THEN
		popupTON2(IN:=FALSE);
		popupStep:=11;
	END_IF
11:
	IF bSendCondition THEN
		popupStep:=12;
	END_IF
	popupTON1(IN:=FALSE);
12:
	//popupTON1(IN:=NOT popupTON1.Q,PT:=T#10MS);
	popupTON1(IN:=NOT popupTON1.Q,PT:=TO_TIME(nQueueInterval));
	IF popupTON1.Q THEN
		popupStep:=0;
	END_IF
END_CASE
END_METHOD

METHOD ReadRTD1 : BOOL
VAR_INPUT
END_VAR
PLC_Chiller.appendSend(16#CA,16#00,16#01,16#20,16#00,16#DE,0,0,0,0,0,0,0,0,0,0,0,0,0,0,10);// 读进水温度
END_METHOD

METHOD ReadRTD2 : BOOL
VAR_INPUT
END_VAR
PLC_Chiller.appendSend(16#CA,16#00,16#01,16#21,16#00,16#DD,0,0,0,0,0,0,0,0,0,0,0,0,0,0,10);// 读RTD2 出水温度
END_METHOD

METHOD ReadState : BOOL
VAR_INPUT
END_VAR
PLC_Chiller.appendSend(16#CA,16#00,16#01,16#09,16#00,16#F5,0,0,0,0,0,0,0,0,0,0,0,0,0,0,10);// 读状态
END_METHOD

METHOD PRIVATE sendData : BOOL
VAR_INPUT
	dataStruct	:struct_byte;
END_VAR
VAR
	str1:STRING;
END_VAR
IF bSendCondition AND bEnable THEN
	tcpipSendData.b1	:=dataStruct.b1;
	tcpipSendData.b2	:=dataStruct.b2;
	tcpipSendData.b3	:=dataStruct.b3;
	tcpipSendData.b4	:=dataStruct.b4;
	tcpipSendData.b5	:=dataStruct.b5;
	tcpipSendData.b6	:=dataStruct.b6;
	tcpipSendData.b7	:=dataStruct.b7;
	tcpipSendData.b8	:=dataStruct.b8;
	tcpipSendData.b9	:=dataStruct.b9;
	tcpipSendData.b10	:=dataStruct.b10;
	tcpipSendData.b11	:=dataStruct.b11;
	tcpipSendData.b12	:=dataStruct.b12;
	tcpipSendData.b13	:=dataStruct.b13;
	tcpipSendData.b14	:=dataStruct.b14;
	tcpipSendData.b15	:=dataStruct.b15;
	tcpipSendData.b16	:=dataStruct.b16;
	tcpipSendData.b17	:=dataStruct.b17;
	tcpipSendData.b18	:=dataStruct.b18;
	tcpipSendData.b19	:=dataStruct.b19;
	tcpipSendData.b20	:=dataStruct.b20;
	
	CASE nSocketType OF
	0://TCPIP server
		tcpipSendDataBuff_Server:=tcpipSendData;
		tcpipSendData:=tcpipSendDataClear;	
		tcpipServer.bSend:=TRUE;
	1://TCPIP client
		tcpipSendDataBuff_Client:=tcpipSendData;
		tcpipSendData:=tcpipSendDataClear;	
		tcpipClient.bSend:=TRUE;
	END_CASE
	
	FOR logHandleArray_index:=1 TO logHandleArrayLength DO
		CASE nSocketType OF
		0://TCPIP server
			str1:=CONCAT(str1,BYTE_TO_HEXSTR(tcpipSendDataBuff_Server.b1,2,FALSE));
			str1:=CONCAT(str1,' ');
			str1:=CONCAT(str1,BYTE_TO_HEXSTR(tcpipSendDataBuff_Server.b2,2,FALSE));
			str1:=CONCAT(str1,' ');
			str1:=CONCAT(str1,BYTE_TO_HEXSTR(tcpipSendDataBuff_Server.b3,2,FALSE));
			str1:=CONCAT(str1,' ');
			str1:=CONCAT(str1,BYTE_TO_HEXSTR(tcpipSendDataBuff_Server.b4,2,FALSE));
			str1:=CONCAT(str1,' ');
			str1:=CONCAT(str1,BYTE_TO_HEXSTR(tcpipSendDataBuff_Server.b5,2,FALSE));
			str1:=CONCAT(str1,' ');
			str1:=CONCAT(str1,BYTE_TO_HEXSTR(tcpipSendDataBuff_Server.b6,2,FALSE));
			str1:=CONCAT(str1,' ');
			str1:=CONCAT(str1,BYTE_TO_HEXSTR(tcpipSendDataBuff_Server.b7,2,FALSE));
			str1:=CONCAT(str1,' ');
			str1:=CONCAT(str1,BYTE_TO_HEXSTR(tcpipSendDataBuff_Server.b8,2,FALSE));
			str1:=CONCAT(str1,' ');
			str1:=CONCAT(str1,BYTE_TO_HEXSTR(tcpipSendDataBuff_Server.b9,2,FALSE));
			str1:=CONCAT(str1,' ');
			str1:=CONCAT(str1,BYTE_TO_HEXSTR(tcpipSendDataBuff_Server.b10,2,FALSE));
			str1:=CONCAT(str1,' ');
			str1:=CONCAT(str1,BYTE_TO_HEXSTR(tcpipSendDataBuff_Server.b11,2,FALSE));
			str1:=CONCAT(str1,' ');
			str1:=CONCAT(str1,BYTE_TO_HEXSTR(tcpipSendDataBuff_Server.b12,2,FALSE));
			str1:=CONCAT(str1,' ');
			str1:=CONCAT(str1,BYTE_TO_HEXSTR(tcpipSendDataBuff_Server.b13,2,FALSE));
			str1:=CONCAT(str1,' ');
			str1:=CONCAT(str1,BYTE_TO_HEXSTR(tcpipSendDataBuff_Server.b14,2,FALSE));
			str1:=CONCAT(str1,' ');
			str1:=CONCAT(str1,BYTE_TO_HEXSTR(tcpipSendDataBuff_Server.b15,2,FALSE));
			str1:=CONCAT(str1,' ');
			str1:=CONCAT(str1,BYTE_TO_HEXSTR(tcpipSendDataBuff_Server.b16,2,FALSE));
			str1:=CONCAT(str1,' ');
			str1:=CONCAT(str1,BYTE_TO_HEXSTR(tcpipSendDataBuff_Server.b17,2,FALSE));
			str1:=CONCAT(str1,' ');
			str1:=CONCAT(str1,BYTE_TO_HEXSTR(tcpipSendDataBuff_Server.b18,2,FALSE));
			str1:=CONCAT(str1,' ');
			str1:=CONCAT(str1,BYTE_TO_HEXSTR(tcpipSendDataBuff_Server.b19,2,FALSE));
			str1:=CONCAT(str1,' ');
			str1:=CONCAT(str1,BYTE_TO_HEXSTR(tcpipSendDataBuff_Server.b20,2,FALSE));
			logHandleArray[logHandleArray_index]^.append(CONCAT(CONCAT(CONCAT('Send To ', sTerminalName), ' -- '),str1));
		1://TCPIP client
			str1:=CONCAT(str1,' ');
			str1:=CONCAT(str1,BYTE_TO_HEXSTR(tcpipSendDataBuff_Client.b1,2,FALSE));
			str1:=CONCAT(str1,' ');
			str1:=CONCAT(str1,BYTE_TO_HEXSTR(tcpipSendDataBuff_Client.b2,2,FALSE));
			str1:=CONCAT(str1,' ');
			str1:=CONCAT(str1,BYTE_TO_HEXSTR(tcpipSendDataBuff_Client.b3,2,FALSE));
			str1:=CONCAT(str1,' ');
			str1:=CONCAT(str1,BYTE_TO_HEXSTR(tcpipSendDataBuff_Client.b4,2,FALSE));
			str1:=CONCAT(str1,' ');
			str1:=CONCAT(str1,BYTE_TO_HEXSTR(tcpipSendDataBuff_Client.b5,2,FALSE));
			str1:=CONCAT(str1,' ');
			str1:=CONCAT(str1,BYTE_TO_HEXSTR(tcpipSendDataBuff_Client.b6,2,FALSE));
			str1:=CONCAT(str1,' ');
			str1:=CONCAT(str1,BYTE_TO_HEXSTR(tcpipSendDataBuff_Client.b7,2,FALSE));
			str1:=CONCAT(str1,' ');
			str1:=CONCAT(str1,BYTE_TO_HEXSTR(tcpipSendDataBuff_Client.b8,2,FALSE));
			str1:=CONCAT(str1,' ');
			str1:=CONCAT(str1,BYTE_TO_HEXSTR(tcpipSendDataBuff_Client.b9,2,FALSE));
			str1:=CONCAT(str1,' ');
			str1:=CONCAT(str1,BYTE_TO_HEXSTR(tcpipSendDataBuff_Client.b10,2,FALSE));
			str1:=CONCAT(str1,' ');
			str1:=CONCAT(str1,BYTE_TO_HEXSTR(tcpipSendDataBuff_Client.b11,2,FALSE));
			str1:=CONCAT(str1,' ');
			str1:=CONCAT(str1,BYTE_TO_HEXSTR(tcpipSendDataBuff_Client.b12,2,FALSE));
			str1:=CONCAT(str1,' ');
			str1:=CONCAT(str1,BYTE_TO_HEXSTR(tcpipSendDataBuff_Client.b13,2,FALSE));
			str1:=CONCAT(str1,' ');
			str1:=CONCAT(str1,BYTE_TO_HEXSTR(tcpipSendDataBuff_Client.b14,2,FALSE));
			str1:=CONCAT(str1,' ');
			str1:=CONCAT(str1,BYTE_TO_HEXSTR(tcpipSendDataBuff_Client.b15,2,FALSE));
			str1:=CONCAT(str1,' ');
			str1:=CONCAT(str1,BYTE_TO_HEXSTR(tcpipSendDataBuff_Client.b16,2,FALSE));
			str1:=CONCAT(str1,' ');
			str1:=CONCAT(str1,BYTE_TO_HEXSTR(tcpipSendDataBuff_Client.b17,2,FALSE));
			str1:=CONCAT(str1,' ');
			str1:=CONCAT(str1,BYTE_TO_HEXSTR(tcpipSendDataBuff_Client.b18,2,FALSE));
			str1:=CONCAT(str1,' ');
			str1:=CONCAT(str1,BYTE_TO_HEXSTR(tcpipSendDataBuff_Client.b19,2,FALSE));
			str1:=CONCAT(str1,' ');
			str1:=CONCAT(str1,BYTE_TO_HEXSTR(tcpipSendDataBuff_Client.b20,2,FALSE));
			logHandleArray[logHandleArray_index]^.append(CONCAT(CONCAT(CONCAT('Send To ', sTerminalName), ' -- '),str1));
		END_CASE
	END_FOR
END_IF
END_METHOD

METHOD WriteStart : BOOL
VAR_INPUT
END_VAR
PLC_Chiller.appendSend(16#CA,16#00,16#01,16#81,16#08,16#01,16#02,16#02,16#02,16#02,16#02,16#02,16#02,16#66,0,0,0,0,0,0,14);// 开机
END_METHOD

METHOD WriteStop : BOOL
VAR_INPUT
END_VAR
PLC_Chiller.appendSend(16#CA,16#00,16#01,16#81,16#08,16#00,16#02,16#02,16#02,16#02,16#02,16#02,16#02,16#67,0,0,0,0,0,0,14);// 开机
END_METHOD

METHOD WriteTemperature : BOOL
VAR_INPUT
	setpointVal:REAL;
END_VAR
VAR
	valTemp:INT;
	valTempH:INT;
	valTempL:INT;
	checkSum:INT;
END_VAR
valTemp:=REAL_TO_INT(setpointVal*10);
valTempH:=valTemp/256;
valTempL:=valTemp MOD 256;
checkSum:=255-(1+240+2+valTempH+valTempL);
PLC_Chiller.readSetAckFlag:=FALSE;
PLC_Chiller.appendSend(16#CA,16#00,16#01,16#F0,16#02,INT_TO_BYTE(valTempH),INT_TO_BYTE(valTempL),INT_TO_BYTE(checkSum),0,0,0,0,0,0,0,0,0,0,0,0,8);// 设定参数
END_METHOD

END_PROGRAM

// ---- POUs/BaseModule/ActionModule/ARMModule/ARMModule.TcPOU
(*
--报错编号0: 无报错
--报错编号1: IN Error
--报错编号2: HOME Error
*)
FUNCTION_BLOCK ARMModule
VAR_IN_OUT
	WarmHMI					:WARMStruct;
	NoteHMI					:NoteStruct;
	operatorLog				:printLogModule_EX;
END_VAR
VAR_INPUT
	HMIItf						:ARMModuleHMI;// 每个ARM对象都关联了一个HMI
	armType						:ARMType:=ARMType_SinSun;// 设置ARM的类型, 可通过该变量修改具体发送的协议内容、、
	
	real_TimeMonitor			:BOOL:=TRUE;//实时状态检测
	
	IN							:BOOL:=FALSE;// 进信号
	INCondition					:BOOL:=TRUE;//  进信号条件
	HOME						:BOOL:=FALSE;// 回触发信号
	HOMECondition				:BOOL:=TRUE;// 回启停条件
	
	JOG							:BOOL:=FALSE;// 点动发信号
	
	readCondition				:BOOL:=TRUE;// 循环读取状态条件
	
	JOGCondition				:BOOL:=TRUE;// 点动启停条件
	reset						:BOOL:=FALSE;//复位信号
	stop						:BOOL:=FALSE;//停止信号
	power						:BOOL:=TRUE;// ARM动作后是否关闭继电器得电状态, TRUE--保持得电,FALSE--断开得电
	enable						:BOOL:=TRUE;//ARM禁用条件
	//ctrlMode					:ControlMode:=ControlMode.eManualCtrMode;//eManualCtrMode or eAutoCtrMode
	hmiEN						:BOOL:=TRUE;//HMI 启用条件
	setpos						:DINT:=8900;// 位置设定
	setvel						:DINT:=10;// 速度设定
	
	jogsetDir					:BOOL:=FALSE;// 方向设定、、 点动设置慎用；
	jogsetlen					:DINT:=1;// 寸动设定、、 点动设置慎用
	minPos						:INT:=0;
	maxPos						:INT:=9000;
	errorDelayTime				:TIME:=T#30S;//ARM感应器感应超时
	//doneDelayTimeShort		:TIME:=T#100MS;//ARM感应到位延时---取消使用
	//doneDelayTimeLong			:TIME:=T#500MS;//无ARM感应到位延时---取消使用
	doneDelayTimeShortIN		:TIME:=T#100MS;//ARM感应到位延时_伸出
	doneDelayTimeShortHOME		:TIME:=T#100MS;//ARM感应到位延时_收回
	doneDelayTimeLongIN			:TIME:=T#500MS;//无ARM感应到位延时_伸出
	doneDelayTimeLongHOME		:TIME:=T#500MS;//无ARM感应到位延时_收回
	errorID						:UDINT:=0;//ARM错误报警分配的起始ID
	nameTXT						:STRING(255):='';//ARM名字
	
	INAprSw						:BOOL:=FALSE;//ARM伸出感应器信号,需要链接到实际的IO点
	HOMEAprSw					:BOOL:=FALSE;//ARM收回感应器信号,需要链接到实际的IO点
	enableINAprSw				:BOOL:=TRUE;//启用伸出感应器,针对只有一个传感器的ARM
	enableHOMEAprSw				:BOOL:=TRUE;//启用收回感应器,针对只有一个传感器的ARM
	noteWTXT_IN					:WSTRING(255):="";//ARM伸出动作NoteTXT 中文
	noteWTXT_HOME				:WSTRING(255):="";//ARM缩回动作NoteTXT 中文
END_VAR
VAR_OUTPUT
	INRelay					:BOOL:=FALSE;//ARM伸出执行继电器,需要链接到实际的IO点
	HOMERelay				:BOOL:=FALSE;//ARM收回执行继电器,需要链接到实际的IO点
	note_IN					:BOOL:=FALSE;// 操作提示：true 伸出、打开执行无法下发
	note_HOME				:BOOL:=FALSE;// 操作提示：true 缩回、关闭执行无法下发
	note_JOG				:BOOL:=FALSE;// 操作提示：true 缩回、关闭执行无法下发
	busy					:BOOL;// ARM动作Busy状态
	done					:BOOL;// ARM动作Done状态
	INdone					:BOOL;// ARM动作伸出完成
	HOMEdone				:BOOL;// ARM动作收回完成
	readdone				:BOOL;// ARM状态完成
	readbusy				:BOOL;
	readerror				:BOOL;
	error					:BOOL;//ARM动作error状态
	errID					:UDINT;//ARM动作errID
	errTXT					:STRING(255):='';//ARM动作errTXT
	errWTXT					:WSTRING(255):="";//ARM动作errTXT 中文
	notRun					:BOOL;
	actpos					:INT;
	jogBusy					:BOOL;
END_VAR
	
VAR
	firstPower				:BOOL:=TRUE;
	firstPowerTON			:TON;
	readAndWriteLock		:BOOL;
	INErrorDelayTon			:Ton;
	INDoneDelayTon			:Ton;
	HOMEErrorDelayTon		:Ton;
	HOMEDoneDelayTon		:Ton;
	
	INTrigRAlc			:R_Trig;//上升沿触发
	
	INTrigR1				:R_Trig;//上升沿触发
	HOMETrigR1			:R_Trig;//上升沿触发
	resetTrigR1				:R_Trig;//上升沿触发
	stopTrigR1				:R_Trig;//上升沿触发
	powerTrigR1				:R_Trig;//上升沿触发
	
	INStep					:UINT:=0;
	HOMEStep				:UINT:=0;
	errorStep				:UINT:=0;
	readStep				:UINT:=0;
	
	notBusyMonitorDelayTon:TON;//动作不切换时，延迟检测
	notBusyMonitorDelayTime:TIME:=T#2S;//动作不切换延迟检测时间
	noteTON_P:tON;            // 操作提示标志位延时继电器
	noteTON_N:tON;            // 操作提示标志位延时继电器
	noteRTrig_P:R_TRIG;          // 操作提示
	noteRTrig_N:R_TRIG;          // 操作提示
	INcheckDelayTime	:TON; // 输出到输入检测时间
	INcheckDelayTimeS	:TIME; // 输出到输入检测时间
	INcheckRtrig:R_TRIG;     // 输出到输入检测
	HOMEcheckDelayTime	:TON; // 输出到输入检测时间
	HOMEcheckDelayTimeS	:TIME; // 输出到输入检测时间
	HOMEcheckRtrig:R_TRIG;     // 输出到输入检测
	
	IndelaycheckTON:TON;
	HomedelaycheckTON:TON;
	IndelaycheckTime:TIME:=T#100MS;
	HomedelaycheckTime:TIME:=T#100MS;
	
	readTon1:TON;
	readTon2:TON;
	
	t1:TON;
	jogResetTON:TON;
	jogResetTime:DINT;
END_VAR

Init_ACT();
Error_ACT();
IN_ACT();
HOME_ACT();
Reset_ACT();
Read_ACT();
Error_ACT();
RealMonitor_ACT();
//		INend:=TRUE;
//		firstPower:=TRUE;
//	END_IF
//	IF HOMEAprSw AND NOT INAprSw THEN
//		HOMEract:=TRUE;
//		firstPower:=TRUE;
//	END_IF
//	IF (NOT INAprSw) AND (NOT HOMEAprSw) THEN
//		errorStep:=3;
//	END_IF
//	IF (INAprSw) AND (HOMEAprSw) THEN
//		errorStep:=3;
//	END_IF
//END_IF

